KUKA KRL program: MyProgram_246().src

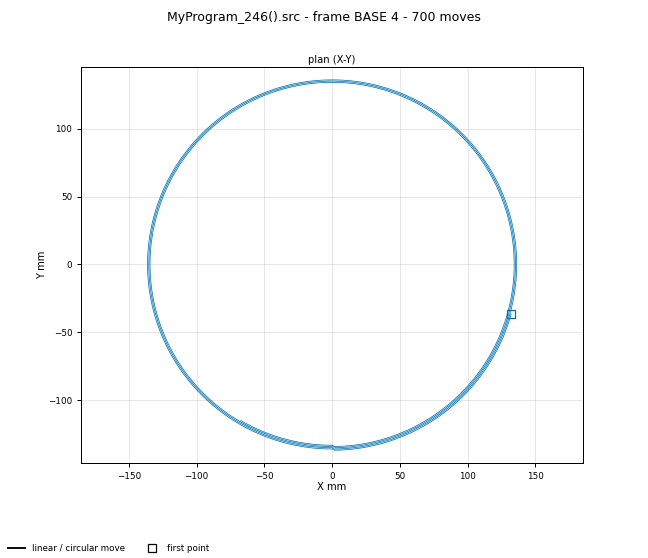
[picture p0: tool path of MyProgram_246().src in frame BASE 4, 700 of 700 moves have a stored position in this frame; points joined in program order, loops and branches not executed]
&ACCESS RVP
&REL 1
&PARAM TEMPLATE = C:\KRC\Roboter\Template\vorgabe
&PARAM EDITMASK = *
DEF MyProgram_246()
; ---- Setting reference (Base) ----
$BASE = BASE_DATA[4]

; --------------------------
; ---- Setting tool (TCP) ----
$TOOL = TOOL_DATA[3]
; --------------------------

$VEL.CP = VEL_APROX_PRINT
Startdeposition()
$VEL.CP = VEL_PRINT
LIN {X 132.0925,Y -36.5753,Z 163,A -18.1429,B 22.0609,C -0.8427,E1 22.2299,E2 825.7735} C_DIS
LIN {X 131.1106,Y -39.9509,Z 163,A -19.472,B 22.0608,C -0.8452,E1 22.2288,E2 827.0873} C_DIS
LIN {X 130.1347,Y -43.0241,Z 163,A -20.8856,B 22.061,C -0.8377,E1 22.2276,E2 828.5116} C_DIS
LIN {X 129.0285,Y -46.2357,Z 163,A -22.4856,B 22.0615,C -0.8242,E1 22.2261,E2 830.1371} C_DIS
LIN {X 126.7894,Y -52.0684,Z 163,A -24.8697,B 22.0615,C -0.8276,E1 22.2237,E2 832.4969} C_DIS
LIN {X 124.8368,Y -56.5884,Z 163,A -27.0477,B 22.0618,C -0.8153,E1 22.2212,E2 834.6937} C_DIS
LIN {X 123.0791,Y -60.313,Z 163,A -28.6428,B 22.0618,C -0.8166,E1 22.2193,E2 836.2756} C_DIS
LIN {X 121.472,Y -63.4871,Z 163,A -29.8971,B 22.0615,C -0.824,E1 22.2177,E2 837.5026} C_DIS
LIN {X 119.8871,Y -66.435,Z 163,A -31.5668,B 22.0622,C -0.8061,E1 22.2155,E2 839.2096} C_DIS
LIN {X 117.7011,Y -70.2353,Z 163,A -33.2997,B 22.0622,C -0.8059,E1 22.213,E2 840.9328} C_DIS
LIN {X 115.1668,Y -74.3185,Z 163,A -35.4245,B 22.0626,C -0.7943,E1 22.2099,E2 843.0759} C_DIS
LIN {X 113.0013,Y -77.5709,Z 163,A -36.9832,B 22.0626,C -0.7936,E1 22.2074,E2 844.6278} C_DIS
LIN {X 110.6195,Y -80.9316,Z 163,A -38.7434,B 22.0628,C -0.7869,E1 22.2045,E2 846.3958} C_DIS
LIN {X 108.0525,Y -84.3289,Z 163,A -40.5478,B 22.063,C -0.7809,E1 22.2015,E2 848.2063} C_DIS
LIN {X 105.289,Y -87.7551,Z 163,A -42.3883,B 22.0632,C -0.7761,E1 22.1982,E2 850.0499} C_DIS
LIN {X 102.3699,Y -91.1433,Z 163,A -44.2158,B 22.0632,C -0.7734,E1 22.1948,E2 851.875} C_DIS
LIN {X 99.5765,Y -94.1865,Z 163,A -45.9214,B 22.0634,C -0.7701,E1 22.1916,E2 853.5806} C_DIS
LIN {X 96.3351,Y -97.4998,Z 163,A -47.8615,B 22.0635,C -0.7653,E1 22.1878,E2 855.524} C_DIS
LIN {X 93.0592,Y -100.6314,Z 163,A -49.7722,B 22.0637,C -0.76,E1 22.1839,E2 857.4397} C_DIS
LIN {X 89.8698,Y -103.4894,Z 163,A -51.5288,B 22.0637,C -0.7576,E1 22.1802,E2 859.1947} C_DIS
LIN {X 86.486,Y -106.3335,Z 163,A -53.3585,B 22.0639,C -0.7544,E1 22.1762,E2 861.0248} C_DIS
LIN {X 82.9341,Y -109.1267,Z 163,A -55.2607,B 22.0641,C -0.7497,E1 22.172,E2 862.9314} C_DIS
LIN {X 79.2487,Y -111.8314,Z 163,A -57.1564,B 22.0641,C -0.7466,E1 22.1677,E2 864.8278} C_DIS
LIN {X 75.5656,Y -114.3522,Z 163,A -58.996,B 22.0642,C -0.7442,E1 22.1635,E2 866.6666} C_DIS
LIN {X 71.7824,Y -116.764,Z 163,A -60.8265,B 22.0642,C -0.7429,E1 22.1592,E2 868.4939} C_DIS
LIN {X 68.0323,Y -118.9881,Z 163,A -62.6432,B 22.0644,C -0.7399,E1 22.1548,E2 870.3122} C_DIS
LIN {X 64.8491,Y -120.7524,Z 163,A -64.145,B 22.0644,C -0.7382,E1 22.1511,E2 871.8134} C_DIS
LIN {X 59.748,Y -123.356,Z 163,A -66.6031,B 22.0646,C -0.7311,E1 22.1449,E2 874.2826} C_DIS
LIN {X 56.2308,Y -124.9967,Z 163,A -67.9718,B 22.0643,C -0.7412,E1 22.1415,E2 875.6207} C_DIS
LIN {X 51.2868,Y -127.105,Z 163,A -71.1817,B 22.0659,C -0.691,E1 22.1329,E2 878.9552} C_DIS
LIN {X 45.3554,Y -129.3412,Z 163,A -73.034,B 22.0648,C -0.7263,E1 22.1283,E2 880.7095} C_DIS
LIN {X 42.0092,Y -130.4659,Z 163,A -74.4413,B 22.0648,C -0.7278,E1 22.1246,E2 882.1096} C_DIS
LIN {X 38.6726,Y -131.4933,Z 163,A -75.8536,B 22.0648,C -0.7285,E1 22.1208,E2 883.5172} C_DIS
LIN {X 35.3588,Y -132.4228,Z 163,A -77.3415,B 22.0648,C -0.7246,E1 22.1168,E2 885.0128} C_DIS
LIN {X 31.7726,Y -133.3292,Z 163,A -78.9793,B 22.065,C -0.7186,E1 22.1123,E2 886.6637} C_DIS
LIN {X 27.2389,Y -134.3284,Z 163,A -81.3195,B 22.0657,C -0.6977,E1 22.1058,E2 889.0561} C_DIS
LIN {X 22.8624,Y -135.1425,Z 163,A -82.6671,B 22.065,C -0.721,E1 22.1023,E2 890.3401} C_DIS
LIN {X 19.2743,Y -135.7004,Z 163,A -84.1486,B 22.065,C -0.7217,E1 22.0982,E2 891.8181} C_DIS
LIN {X 14.7543,Y -136.266,Z 163,A -85.8072,B 22.0646,C -0.7324,E1 22.0937,E2 893.4468} C_DIS
LIN {X 8.5698,Y -136.7944,Z 163,A -88.7021,B 22.0651,C -0.7167,E1 22.0855,E2 896.3818} C_DIS
LIN {X 1.7574,Y -137.0523,Z 163,A -91.484,B 22.0651,C -0.719,E1 22.0778,E2 899.1566} C_DIS
LIN {X 1.7574,Y -137.0523,Z 163,A -91.484,B 22.0651,C -0.719,E1 22.0778,E2 899.1566} C_DIS
Enddeposition()
LIN {X 0.9573,Y -136.1368,Z 163,A -91.0711,B 20.8323,C -0.5633,E1 20.8415,E2 899.0478} C_DIS
Startdeposition()
$VEL.CP = VEL_PRINT
LIN {X 5.9809,Y -136.0119,Z 163,A -88.7973,B 20.8321,C -0.571,E1 20.8479,E2 896.7528} C_DIS
LIN {X 12.7142,Y -135.5469,Z 163,A -85.8042,B 20.8319,C -0.5792,E1 20.8563,E2 893.7385} C_DIS
LIN {X 16.2786,Y -135.1649,Z 163,A -84.4391,B 20.8321,C -0.5735,E1 20.86,E2 892.3908} C_DIS
LIN {X 19.3754,Y -134.7557,Z 163,A -83.0441,B 20.8319,C -0.578,E1 20.8639,E2 890.9845} C_DIS
LIN {X 23.679,Y -134.0667,Z 163,A -81.084,B 20.8318,C -0.5852,E1 20.8693,E2 889.007} C_DIS
LIN {X 28.5269,Y -133.1192,Z 163,A -79.1368,B 20.8318,C -0.5808,E1 20.8746,E2 887.075} C_DIS
LIN {X 31.9197,Y -132.3465,Z 163,A -77.6987,B 20.8318,C -0.581,E1 20.8785,E2 885.6389} C_DIS
LIN {X 35.3669,Y -131.4676,Z 163,A -76.2581,B 20.8319,C -0.5798,E1 20.8824,E2 884.2042} C_DIS
LIN {X 38.3717,Y -130.6219,Z 163,A -74.9511,B 20.8319,C -0.5809,E1 20.8859,E2 882.8968} C_DIS
LIN {X 41.669,Y -129.6079,Z 163,A -73.4798,B 20.8319,C -0.5835,E1 20.8899,E2 881.4216} C_DIS
LIN {X 44.6107,Y -128.6247,Z 163,A -71.8069,B 20.8313,C -0.6022,E1 20.8944,E2 879.7003} C_DIS
LIN {X 48.0166,Y -127.3927,Z 163,A -70.62,B 20.8317,C -0.5884,E1 20.8974,E2 878.5551} C_DIS
LIN {X 51.6805,Y -125.9533,Z 163,A -68.7633,B 20.8314,C -0.6,E1 20.9023,E2 876.6711} C_DIS
LIN {X 56.0611,Y -124.0638,Z 163,A -67.0228,B 20.8316,C -0.5905,E1 20.9066,E2 874.9626} C_DIS
LIN {X 59.4493,Y -122.4779,Z 163,A -65.1913,B 20.8312,C -0.605,E1 20.9113,E2 873.0964} C_DIS
LIN {X 66.6727,Y -118.7,Z 163,A -62.3065,B 20.8318,C -0.5851,E1 20.9183,E2 870.2774} C_DIS
LIN {X 70.855,Y -116.2526,Z 163,A -59.915,B 20.8312,C -0.6052,E1 20.9242,E2 867.8384} C_DIS
LIN {X 74.3486,Y -114.0495,Z 163,A -58.1316,B 20.8311,C -0.6106,E1 20.9284,E2 866.0469} C_DIS
LIN {X 78.1376,Y -111.4882,Z 163,A -56.1985,B 20.8309,C -0.6148,E1 20.9328,E2 864.1102} C_DIS
LIN {X 81.7741,Y -108.8486,Z 163,A -54.3187,B 20.8309,C -0.6181,E1 20.937,E2 862.2294} C_DIS
LIN {X 85.3978,Y -106.0291,Z 163,A -52.427,B 20.8308,C -0.6203,E1 20.9412,E2 860.3401} C_DIS
LIN {X 88.777,Y -103.2162,Z 163,A -50.5846,B 20.8307,C -0.624,E1 20.9451,E2 858.4961} C_DIS
LIN {X 92.0524,Y -100.306,Z 163,A -48.754,B 20.8306,C -0.6276,E1 20.9489,E2 856.6645} C_DIS
LIN {X 95.2418,Y -97.2828,Z 163,A -46.9125,B 20.8305,C -0.6316,E1 20.9526,E2 854.8213} C_DIS
LIN {X 98.3507,Y -94.1387,Z 163,A -45.0732,B 20.8304,C -0.6351,E1 20.9562,E2 852.9819} C_DIS
LIN {X 101.3955,Y -90.8509,Z 163,A -43.1907,B 20.8302,C -0.6396,E1 20.9597,E2 851.097} C_DIS
LIN {X 104.3997,Y -87.3822,Z 163,A -41.3152,B 20.8302,C -0.6418,E1 20.9631,E2 849.2256} C_DIS
LIN {X 107.1983,Y -83.9256,Z 163,A -39.4537,B 20.83,C -0.6462,E1 20.9664,E2 847.3625} C_DIS
LIN {X 109.7297,Y -80.5874,Z 163,A -37.6614,B 20.8299,C -0.6523,E1 20.9694,E2 845.5637} C_DIS
LIN {X 113.5217,Y -75.1515,Z 163,A -34.9433,B 20.8297,C -0.6565,E1 20.9737,E2 842.8502} C_DIS
LIN {X 117.1344,Y -69.3873,Z 163,A -32.2387,B 20.8297,C -0.6569,E1 20.9776,E2 840.1614} C_DIS
LIN {X 119.8054,Y -64.6659,Z 163,A -29.8094,B 20.8293,C -0.6705,E1 20.9809,E2 837.7095} C_DIS
LIN {X 121.5803,Y -61.2612,Z 163,A -28.2663,B 20.8293,C -0.6717,E1 20.9829,E2 836.1731} C_DIS
LIN {X 123.175,Y -57.9906,Z 163,A -26.752,B 20.8292,C -0.6754,E1 20.9847,E2 834.6584} C_DIS
LIN {X 124.9426,Y -54.0718,Z 163,A -24.9018,B 20.8289,C -0.6828,E1 20.9868,E2 832.7998} C_DIS
LIN {X 128.2312,Y -45.732,Z 163,A -21.212,B 20.8287,C -0.6902,E1 20.9905,E2 829.1146} C_DIS
LIN {X 129.623,Y -41.6217,Z 163,A -19.638,B 20.8289,C -0.6837,E1 20.9919,E2 827.5697} C_DIS
LIN {X 130.5484,Y -38.6225,Z 163,A -18.0389,B 20.8283,C -0.7011,E1 20.9932,E2 825.933} C_DIS
LIN {X 131.5669,Y -34.9944,Z 163,A -16.529,B 20.8283,C -0.7024,E1 20.9943,E2 824.43} C_DIS
LIN {X 132.5583,Y -31.0367,Z 163,A -14.8544,B 20.8282,C -0.7057,E1 20.9954,E2 822.758} C_DIS
LIN {X 133.4538,Y -26.9184,Z 163,A -13.0033,B 20.8279,C -0.7151,E1 20.9965,E2 820.894} C_DIS
LIN {X 134.2072,Y -22.8721,Z 163,A -11.2678,B 20.8277,C -0.7207,E1 20.9973,E2 819.1553} C_DIS
LIN {X 134.8677,Y -18.5875,Z 163,A -9.142,B 20.827,C -0.7411,E1 20.9982,E2 816.9878} C_DIS
LIN {X 135.323,Y -14.9104,Z 163,A -8.1608,B 20.8278,C -0.7181,E1 20.9985,E2 816.0779} C_DIS
LIN {X 135.6299,Y -11.7967,Z 163,A -6.6477,B 20.8273,C -0.7318,E1 20.9989,E2 814.5377} C_DIS
LIN {X 135.8901,Y -8.2723,Z 163,A -5.1603,B 20.8272,C -0.7366,E1 20.9992,E2 813.0477} C_DIS
LIN {X 136.1148,Y -2.7468,Z 163,A -2.7081,B 20.8267,C -0.75,E1 20.9994,E2 810.5759} C_DIS
LIN {X 136.1245,Y 2.1662,Z 163,A -0.8222,B 20.8267,C -0.7478,E1 20.9994,E2 808.7098} C_DIS
LIN {X 136.0139,Y 5.9299,Z 163,A 0.9134,B 20.8264,C -0.7601,E1 20.9992,E2 806.9525} C_DIS
LIN {X 135.735,Y 10.5321,Z 163,A 2.7811,B 20.8263,C -0.7627,E1 20.9988,E2 805.091} C_DIS
LIN {X 135.3786,Y 14.3939,Z 163,A 4.3054,B 20.8263,C -0.7627,E1 20.9984,E2 803.5778} C_DIS
LIN {X 134.9328,Y 18.1054,Z 163,A 6.012,B 20.8259,C -0.774,E1 20.9978,E2 801.8519} C_DIS
LIN {X 134.2951,Y 22.3454,Z 163,A 7.6827,B 20.8259,C -0.7732,E1 20.997,E2 800.1955} C_DIS
LIN {X 133.6398,Y 25.982,Z 163,A 9.2348,B 20.8257,C -0.7779,E1 20.9962,E2 798.6414} C_DIS
LIN {X 132.7822,Y 30.0569,Z 163,A 10.9588,B 20.8256,C -0.7819,E1 20.9952,E2 796.9185} C_DIS
LIN {X 131.9441,Y 33.5441,Z 163,A 12.4263,B 20.8255,C -0.7845,E1 20.9942,E2 795.4541} C_DIS
LIN {X 131.0161,Y 37.0048,Z 163,A 13.9109,B 20.8254,C -0.7879,E1 20.9931,E2 793.9704} C_DIS
LIN {X 129.2131,Y 42.8767,Z 163,A 16.9254,B 20.8243,C -0.8163,E1 20.9905,E2 790.8976} C_DIS
LIN {X 127.8235,Y 46.8625,Z 163,A 18.2224,B 20.825,C -0.7984,E1 20.9894,E2 789.6593} C_DIS
LIN {X 126.1483,Y 51.1969,Z 163,A 20.2191,B 20.8247,C -0.8061,E1 20.9873,E2 787.6547} C_DIS
LIN {X 124.8548,Y 54.2749,Z 163,A 21.5923,B 20.8247,C -0.8086,E1 20.9858,E2 786.2838} C_DIS
LIN {X 123.179,Y 57.9823,Z 163,A 23.3882,B 20.8243,C -0.8174,E1 20.9837,E2 784.4753} C_DIS
LIN {X 121.3746,Y 61.6653,Z 163,A 25.0582,B 20.8243,C -0.8195,E1 20.9816,E2 782.8101} C_DIS
LIN {X 119.498,Y 65.2317,Z 163,A 26.7749,B 20.824,C -0.8251,E1 20.9793,E2 781.0889} C_DIS
LIN {X 117.2985,Y 69.1089,Z 163,A 28.618,B 20.8239,C -0.8285,E1 20.9768,E2 779.2479} C_DIS
LIN {X 114.955,Y 72.9409,Z 163,A 30.4779,B 20.8237,C -0.832,E1 20.974,E2 777.3897} C_DIS
LIN {X 112.5835,Y 76.5505,Z 163,A 33.224,B 20.8218,C -0.881,E1 20.9695,E2 774.5233} C_DIS
LIN {X 108.4547,Y 82.2961,Z 163,A 35.4253,B 20.823,C -0.8512,E1 20.966,E2 772.4183} C_DIS
LIN {X 105.3366,Y 86.2504,Z 163,A 37.38,B 20.8231,C -0.8484,E1 20.9626,E2 770.4824} C_DIS
LIN {X 102.4793,Y 89.6268,Z 163,A 39.4353,B 20.8226,C -0.8619,E1 20.9588,E2 768.401} C_DIS
LIN {X 100.3058,Y 92.0526,Z 163,A 40.4025,B 20.8232,C -0.846,E1 20.9571,E2 767.4835} C_DIS
LIN {X 98.0621,Y 94.4398,Z 163,A 41.985,B 20.8227,C -0.8585,E1 20.954,E2 765.8743} C_DIS
LIN {X 94.9308,Y 97.5868,Z 163,A 43.8663,B 20.8225,C -0.8631,E1 20.9502,E2 763.9898} C_DIS
LIN {X 91.9581,Y 100.3927,Z 163,A 45.5187,B 20.8225,C -0.8634,E1 20.9469,E2 762.3448} C_DIS
LIN {X 88.7505,Y 103.239,Z 163,A 48.4672,B 20.8202,C -0.9208,E1 20.9403,E2 759.2496} C_DIS
LIN {X 82.3061,Y 108.4471,Z 163,A 50.5399,B 20.8226,C -0.8608,E1 20.9361,E2 757.3544} C_DIS
LIN {X 79.4229,Y 110.5759,Z 163,A 52.2003,B 20.8222,C -0.8705,E1 20.9323,E2 755.6742} C_DIS
LIN {X 76.1216,Y 112.8738,Z 163,A 53.9563,B 20.822,C -0.8762,E1 20.9283,E2 753.9094} C_DIS
LIN {X 72.4598,Y 115.2587,Z 163,A 55.8307,B 20.8218,C -0.8807,E1 20.9238,E2 752.0297} C_DIS
LIN {X 68.6015,Y 117.5965,Z 163,A 57.7104,B 20.8218,C -0.8827,E1 20.9193,E2 750.1516} C_DIS
LIN {X 64.807,Y 119.7296,Z 163,A 59.5703,B 20.8216,C -0.8865,E1 20.9148,E2 748.2876} C_DIS
LIN {X 61.5076,Y 121.4549,Z 163,A 61.0638,B 20.8216,C -0.8853,E1 20.9111,E2 746.8028} C_DIS
LIN {X 57.8827,Y 123.2261,Z 163,A 62.8484,B 20.8214,C -0.8913,E1 20.9066,E2 745.007} C_DIS
LIN {X 53.4721,Y 125.2019,Z 163,A 64.7371,B 20.8216,C -0.887,E1 20.9018,E2 743.136} C_DIS
LIN {X 47.2983,Y 127.6618,Z 163,A 67.0639,B 20.8223,C -0.8685,E1 20.8959,E2 740.8675} C_DIS
LIN {X 44.4361,Y 128.6852,Z 163,A 68.7845,B 20.8215,C -0.8896,E1 20.8912,E2 739.092} C_DIS
LIN {X 41.1735,Y 129.7661,Z 163,A 70.2438,B 20.8214,C -0.8914,E1 20.8873,E2 737.631} C_DIS
LIN {X 38.008,Y 130.7284,Z 163,A 71.6147,B 20.8214,C -0.8914,E1 20.8837,E2 736.2629} C_DIS
LIN {X 34.8398,Y 131.6081,Z 163,A 73.039,B 20.8213,C -0.8942,E1 20.8798,E2 734.8335} C_DIS
LIN {X 30.6655,Y 132.6432,Z 163,A 74.8681,B 20.8212,C -0.8961,E1 20.8748,E2 733.0023} C_DIS
LIN {X 26.8947,Y 133.4587,Z 163,A 76.4627,B 20.8212,C -0.8956,E1 20.8705,E2 731.4115} C_DIS
LIN {X 21.3324,Y 134.4607,Z 163,A 78.6958,B 20.8214,C -0.89,E1 20.8644,E2 729.1971} C_DIS
LIN {X 17.5624,Y 135.004,Z 163,A 80.4262,B 20.8212,C -0.8962,E1 20.8596,E2 727.4513} C_DIS
LIN {X 13.5394,Y 135.4677,Z 163,A 82.3449,B 20.8208,C -0.906,E1 20.8542,E2 725.5065} C_DIS
LIN {X 7.7658,Y 135.9213,Z 163,A 84.5265,B 20.8212,C -0.8948,E1 20.8482,E2 723.3577} C_DIS
LIN {X 4.097,Y 136.0804,Z 163,A 86.1427,B 20.8212,C -0.8979,E1 20.8437,E2 721.7334} C_DIS
LIN {X 0.3597,Y 136.1418,Z 163,A 87.9402,B 20.8207,C -0.9076,E1 20.8386,E2 719.9086} C_DIS
LIN {X -5.8293,Y 136.0178,Z 163,A 90.4101,B 20.821,C -0.901,E1 20.8317,E2 717.457} C_DIS
LIN {X -9.9412,Y 135.7781,Z 163,A 91.9998,B 20.8213,C -0.8941,E1 20.8273,E2 715.8861} C_DIS
LIN {X -13.4121,Y 135.4799,Z 163,A 93.6793,B 20.8209,C -0.9028,E1 20.8226,E2 714.1811} C_DIS
LIN {X -17.2844,Y 135.0404,Z 163,A 95.1442,B 20.8213,C -0.8942,E1 20.8186,E2 712.7391} C_DIS
LIN {X -20.8954,Y 134.5284,Z 163,A 96.7643,B 20.8212,C -0.897,E1 20.8141,E2 711.1095} C_DIS
LIN {X -24.8379,Y 133.8585,Z 163,A 98.5198,B 20.8211,C -0.8989,E1 20.8093,E2 709.3464} C_DIS
LIN {X -29.0692,Y 133.0022,Z 163,A 100.138,B 20.8215,C -0.8888,E1 20.8049,E2 707.7542} C_DIS
LIN {X -32.1683,Y 132.2866,Z 163,A 101.5117,B 20.8215,C -0.8892,E1 20.8012,E2 706.3773} C_DIS
LIN {X -35.917,Y 131.3203,Z 163,A 103.8019,B 20.8204,C -0.9163,E1 20.7948,E2 704.0064} C_DIS
LIN {X -40.8106,Y 129.8821,Z 163,A 105.2335,B 20.8217,C -0.8829,E1 20.7912,E2 702.6659} C_DIS
LIN {X -44.8032,Y 128.5579,Z 163,A 107.097,B 20.8217,C -0.8849,E1 20.7862,E2 700.7924} C_DIS
LIN {X -48.3813,Y 127.2561,Z 163,A 109.0164,B 20.8212,C -0.8965,E1 20.7811,E2 698.8355} C_DIS
LIN {X -51.5758,Y 125.9954,Z 163,A 110.1213,B 20.8219,C -0.8799,E1 20.7784,E2 697.7743} C_DIS
LIN {X -54.4325,Y 124.7866,Z 163,A 111.4691,B 20.8219,C -0.8799,E1 20.7749,E2 696.4227} C_DIS
LIN {X -57.5838,Y 123.3643,Z 163,A 113.0577,B 20.8217,C -0.8835,E1 20.7708,E2 694.8192} C_DIS
LIN {X -61.7482,Y 121.3324,Z 163,A 114.8859,B 20.822,C -0.8753,E1 20.7663,E2 693.0083} C_DIS
LIN {X -66.637,Y 118.72,Z 163,A 117.2559,B 20.8221,C -0.873,E1 20.7605,E2 690.6366} C_DIS
LIN {X -70.2398,Y 116.6249,Z 163,A 119.0789,B 20.8221,C -0.8728,E1 20.7561,E2 688.8073} C_DIS
LIN {X -74.0171,Y 114.2647,Z 163,A 121.0574,B 20.8221,C -0.8738,E1 20.7514,E2 686.8183} C_DIS
LIN {X -77.6596,Y 111.8207,Z 163,A 122.9462,B 20.8221,C -0.872,E1 20.7471,E2 684.9266} C_DIS
LIN {X -81.7195,Y 108.8897,Z 163,A 124.9509,B 20.8225,C -0.8634,E1 20.7426,E2 682.9375} C_DIS
LIN {X -85.1756,Y 106.2083,Z 163,A 126.7323,B 20.8228,C -0.8571,E1 20.7387,E2 681.166} C_DIS
LIN {X -88.4711,Y 103.4792,Z 163,A 128.6154,B 20.8228,C -0.8566,E1 20.7347,E2 679.2753} C_DIS
LIN {X -91.8613,Y 100.4817,Z 163,A 130.5003,B 20.823,C -0.8515,E1 20.7308,E2 677.3955} C_DIS
LIN {X -95.0379,Y 97.4828,Z 163,A 132.3997,B 20.823,C -0.8498,E1 20.7269,E2 675.4914} C_DIS
LIN {X -98.2023,Y 94.2939,Z 163,A 134.2528,B 20.8233,C -0.8437,E1 20.7233,E2 673.6457} C_DIS
LIN {X -101.1802,Y 91.0913,Z 163,A 136.1455,B 20.8233,C -0.8414,E1 20.7198,E2 671.7494} C_DIS
LIN {X -105.6974,Y 85.808,Z 163,A 139.025,B 20.8237,C -0.8321,E1 20.7146,E2 668.8801} C_DIS
LIN {X -110.6727,Y 79.2874,Z 163,A 142.9014,B 20.8234,C -0.8406,E1 20.7081,E2 664.9567} C_DIS
LIN {X -113.073,Y 75.8256,Z 163,A 144.0969,B 20.8245,C -0.8118,E1 20.7063,E2 663.8354} C_DIS
LIN {X -114.6408,Y 73.4331,Z 163,A 145.505,B 20.8243,C -0.8169,E1 20.7041,E2 662.4041} C_DIS
LIN {X -117.0187,Y 69.5814,Z 163,A 147.4308,B 20.8245,C -0.8124,E1 20.7014,E2 660.4789} C_DIS
LIN {X -120.983,Y 62.4345,Z 163,A 151.1407,B 20.8245,C -0.8137,E1 20.6964,E2 656.7413} C_DIS
LIN {X -122.5226,Y 59.3561,Z 163,A 152.23,B 20.8251,C -0.7946,E1 20.6951,E2 655.6989} C_DIS
LIN {X -123.6631,Y 56.9376,Z 163,A 153.4169,B 20.8251,C -0.7938,E1 20.6937,E2 654.5062} C_DIS
LIN {X -125.2267,Y 53.4145,Z 163,A 155.2445,B 20.8251,C -0.7975,E1 20.6917,E2 652.6559} C_DIS
LIN {X -126.8586,Y 49.4097,Z 163,A 156.9217,B 20.8254,C -0.7861,E1 20.69,E2 650.9994} C_DIS
LIN {X -128.251,Y 45.6769,Z 163,A 158.6773,B 20.8255,C -0.7842,E1 20.6883,E2 649.2369} C_DIS
LIN {X -129.6144,Y 41.6485,Z 163,A 160.3687,B 20.8258,C -0.7747,E1 20.6868,E2 647.5607} C_DIS
LIN {X -130.7959,Y 37.7774,Z 163,A 162.076,B 20.826,C -0.7696,E1 20.6854,E2 645.8557} C_DIS
LIN {X -131.5688,Y 34.9873,Z 163,A 163.3057,B 20.8261,C -0.7663,E1 20.6846,E2 644.6267} C_DIS
LIN {X -132.4179,Y 31.6236,Z 163,A 164.8344,B 20.8262,C -0.7645,E1 20.6835,E2 643.092} C_DIS
LIN {X -133.3651,Y 27.3547,Z 163,A 166.6594,B 20.8264,C -0.7581,E1 20.6825,E2 641.2719} C_DIS
LIN {X -134.0485,Y 23.781,Z 163,A 168.159,B 20.8266,C -0.752,E1 20.6817,E2 639.7788} C_DIS
LIN {X -134.5945,Y 20.4685,Z 163,A 169.7405,B 20.8266,C -0.7544,E1 20.681,E2 638.1788} C_DIS
LIN {X -135.1778,Y 16.1699,Z 163,A 171.4502,B 20.8269,C -0.7439,E1 20.6804,E2 636.4865} C_DIS
LIN {X -135.5459,Y 12.724,Z 163,A 172.9275,B 20.8271,C -0.74,E1 20.68,E2 635.0093} C_DIS
LIN {X -135.8612,Y 8.7417,Z 163,A 174.6666,B 20.8271,C -0.737,E1 20.6797,E2 633.2658} C_DIS
LIN {X -136.0416,Y 5.2189,Z 163,A 176.1221,B 20.8274,C -0.7311,E1 20.6795,E2 631.8163} C_DIS
LIN {X -136.136,Y 1.4189,Z 163,A 177.7923,B 20.8274,C -0.7289,E1 20.6795,E2 630.14} C_DIS
LIN {X -136.1117,Y -2.9358,Z 163,A 179.6957,B 20.8275,C -0.726,E1 20.6795,E2 628.2307} C_DIS
LIN {X -135.9626,Y -6.9812,Z 163,A -178.7261,B 20.8279,C -0.7155,E1 20.6797,E2 626.6708} C_DIS
LIN {X -135.7132,Y -10.8108,Z 163,A -176.9918,B 20.8279,C -0.7153,E1 20.68,E2 624.9243} C_DIS
LIN {X -135.3431,Y -14.7234,Z 163,A -175.4203,B 20.8282,C -0.7067,E1 20.6805,E2 623.3656} C_DIS
LIN {X -134.8365,Y -18.8103,Z 163,A -173.6236,B 20.8282,C -0.7039,E1 20.6811,E2 621.5636} C_DIS
LIN {X -134.2924,Y -22.3615,Z 163,A -172.1656,B 20.8285,C -0.6969,E1 20.6818,E2 620.1146} C_DIS
LIN {X -133.6825,Y -25.7585,Z 163,A -170.7234,B 20.8286,C -0.692,E1 20.6825,E2 618.6759} C_DIS
LIN {X -133.0247,Y -28.9648,Z 163,A -169.2852,B 20.8286,C -0.6903,E1 20.6833,E2 617.2321} C_DIS
LIN {X -132.2792,Y -32.1988,Z 163,A -167.8427,B 20.8288,C -0.6879,E1 20.6843,E2 615.786} C_DIS
LIN {X -130.7052,Y -38.0869,Z 163,A -165.5601,B 20.8294,C -0.6685,E1 20.6859,E2 613.5422} C_DIS
LIN {X -129.6447,Y -41.5536,Z 163,A -163.7493,B 20.8291,C -0.6757,E1 20.6874,E2 611.6981} C_DIS
LIN {X -128.5232,Y -44.9034,Z 163,A -162.3055,B 20.8293,C -0.6696,E1 20.6887,E2 610.2616} C_DIS
LIN {X -127.4779,Y -47.7891,Z 163,A -160.9544,B 20.8293,C -0.6683,E1 20.69,E2 608.9048} C_DIS
LIN {X -126.1781,Y -51.1229,Z 163,A -159.4282,B 20.8295,C -0.6648,E1 20.6916,E2 607.3782} C_DIS
LIN {X -124.5868,Y -54.8918,Z 163,A -156.808,B 20.8285,C -0.6976,E1 20.6947,E2 604.6472} C_DIS
LIN {X -121.8227,Y -60.7783,Z 163,A -154.9709,B 20.8299,C -0.6521,E1 20.6968,E2 602.9269} C_DIS
LIN {X -120.2522,Y -63.8291,Z 163,A -153.3683,B 20.8298,C -0.6548,E1 20.6989,E2 601.3062} C_DIS
LIN {X -118.4363,Y -67.141,Z 163,A -151.7764,B 20.8299,C -0.6506,E1 20.7011,E2 599.7158} C_DIS
LIN {X -116.1072,Y -71.092,Z 163,A -149.8622,B 20.8301,C -0.6449,E1 20.7038,E2 597.8058} C_DIS
LIN {X -113.7371,Y -74.8252,Z 163,A -147.8731,B 20.8301,C -0.6455,E1 20.7069,E2 595.8027} C_DIS
LIN {X -111.2507,Y -78.4743,Z 163,A -146.1168,B 20.8303,C -0.6365,E1 20.7097,E2 594.0611} C_DIS
LIN {X -108.5291,Y -82.1975,Z 163,A -144.137,B 20.8304,C -0.6334,E1 20.713,E2 592.0784} C_DIS
LIN {X -105.6584,Y -85.8567,Z 163,A -142.225,B 20.8306,C -0.6269,E1 20.7163,E2 590.1739} C_DIS
LIN {X -102.7115,Y -89.3606,Z 163,A -140.4717,B 20.8309,C -0.6151,E1 20.7194,E2 588.4442} C_DIS
LIN {X -100.6359,Y -91.692,Z 163,A -138.9687,B 20.8308,C -0.6202,E1 20.7223,E2 586.9185} C_DIS
LIN {X -97.6641,Y -94.8509,Z 163,A -137.1109,B 20.8308,C -0.6176,E1 20.7259,E2 585.0581} C_DIS
LIN {X -94.4263,Y -98.0752,Z 163,A -135.1682,B 20.831,C -0.6144,E1 20.7297,E2 583.1144} C_DIS
LIN {X -91.1334,Y -101.1424,Z 163,A -132.6379,B 20.8303,C -0.6381,E1 20.7352,E2 580.5049} C_DIS
LIN {X -86.9261,Y -104.7798,Z 163,A -130.9172,B 20.8312,C -0.6068,E1 20.7387,E2 578.8644} C_DIS
LIN {X -83.3708,Y -107.6301,Z 163,A -128.889,B 20.8312,C -0.6081,E1 20.7431,E2 576.8234} C_DIS
LIN {X -79.4778,Y -110.5366,Z 163,A -126.9727,B 20.8314,C -0.599,E1 20.7474,E2 574.9244} C_DIS
LIN {X -75.9559,Y -112.986,Z 163,A -125.0987,B 20.8314,C -0.599,E1 20.7517,E2 573.0428} C_DIS
LIN {X -72.2627,Y -115.3828,Z 163,A -123.239,B 20.8314,C -0.5965,E1 20.7561,E2 571.183} C_DIS
LIN {X -68.5357,Y -117.6348,Z 163,A -121.4131,B 20.8315,C -0.5935,E1 20.7605,E2 569.3587} C_DIS
LIN {X -64.7496,Y -119.7604,Z 163,A -119.5834,B 20.8315,C -0.5911,E1 20.765,E2 567.5293} C_DIS
LIN {X -61.4846,Y -121.4666,Z 163,A -118.1403,B 20.8318,C -0.5845,E1 20.7685,E2 566.1001} C_DIS
LIN {X -58.733,Y -122.8203,Z 163,A -116.766,B 20.8318,C -0.5866,E1 20.772,E2 564.7155} C_DIS
LIN {X -54.9297,Y -124.5699,Z 163,A -114.3782,B 20.831,C -0.6122,E1 20.7783,E2 562.2485} C_DIS
LIN {X -49.9485,Y -126.6492,Z 163,A -112.8635,B 20.832,C -0.5765,E1 20.782,E2 560.8305} C_DIS
LIN {X -45.0737,Y -128.4642,Z 163,A -110.5012,B 20.8318,C -0.5821,E1 20.7882,E2 558.4465} C_DIS
LIN {X -41.3262,Y -129.7173,Z 163,A -108.9279,B 20.832,C -0.5768,E1 20.7924,E2 556.8845} C_DIS
LIN {X -38.1106,Y -130.6983,Z 163,A -107.5176,B 20.832,C -0.5756,E1 20.7962,E2 555.4748} C_DIS
LIN {X -34.8818,Y -131.5969,Z 163,A -106.1032,B 20.832,C -0.5749,E1 20.8,E2 554.0599} C_DIS
LIN {X -31.3815,Y -132.4762,Z 163,A -104.6066,B 20.832,C -0.573,E1 20.804,E2 552.5659} C_DIS
LIN {X -28.0033,Y -133.2323,Z 163,A -102.607,B 20.8314,C -0.5966,E1 20.8097,E2 550.4969} C_DIS
LIN {X -23.7225,Y -134.0589,Z 163,A -101.4698,B 20.8323,C -0.5647,E1 20.8126,E2 549.4482} C_DIS
LIN {X -20.8214,Y -134.5398,Z 163,A -100.0094,B 20.832,C -0.5742,E1 20.8167,E2 547.9593} C_DIS
LIN {X -16.5914,Y -135.1275,Z 163,A -97.9491,B 20.8317,C -0.5857,E1 20.8225,E2 545.8651} C_DIS
LIN {X -13.3298,Y -135.4878,Z 163,A -96.2394,B 20.8313,C -0.6004,E1 20.8273,E2 544.1126} C_DIS
LIN {X -8.2889,Y -135.8891,Z 163,A -94.733,B 20.8321,C -0.5722,E1 20.8313,E2 542.6851} C_DIS
LIN {X -4.6976,Y -136.0619,Z 163,A -92.5718,B 20.8313,C -0.6018,E1 20.8376,E2 540.4403} C_DIS
LIN {X 0.4637,Y -136.1412,Z 163,A -91.0917,B 20.8321,C -0.5707,E1 20.8415,E2 539.0478} C_DIS
LIN {X 0.4637,Y -136.1412,Z 163,A -91.0917,B 20.8321,C -0.5707,E1 20.8415,E2 539.0478} C_DIS
Enddeposition()
LIN {X 0.9493,Y -135.2146,Z 163,A -90.7114,B 19.607,C -0.4067,E1 19.6129,E2 539.0313} C_DIS
Startdeposition()
$VEL.CP = VEL_PRINT
LIN {X -2.1021,Y -135.2045,Z 163,A -92.3957,B 19.6073,C -0.39,E1 19.6081,E2 540.7652} C_DIS
LIN {X -5.3088,Y -135.1165,Z 163,A -93.7552,B 19.6073,C -0.3899,E1 19.6043,E2 542.1254} C_DIS
LIN {X -9.0786,Y -134.9177,Z 163,A -95.339,B 19.6073,C -0.3905,E1 19.5999,E2 543.708} C_DIS
LIN {X -13.0731,Y -134.5873,Z 163,A -97.0415,B 19.6073,C -0.3905,E1 19.5951,E2 545.4115} C_DIS
LIN {X -16.1777,Y -134.2494,Z 163,A -98.3767,B 19.6073,C -0.3902,E1 19.5914,E2 546.7486} C_DIS
LIN {X -19.44,Y -133.8162,Z 163,A -99.8068,B 19.6073,C -0.3891,E1 19.5874,E2 548.1836} C_DIS
LIN {X -23.0371,Y -133.246,Z 163,A -101.3121,B 19.6073,C -0.3911,E1 19.5833,E2 549.6846} C_DIS
LIN {X -27.1167,Y -132.4737,Z 163,A -103.0903,B 19.6073,C -0.3911,E1 19.5784,E2 551.4654} C_DIS
LIN {X -30.8991,Y -131.6452,Z 163,A -104.7215,B 19.6073,C -0.3923,E1 19.574,E2 553.0958} C_DIS
LIN {X -34.053,Y -130.8649,Z 163,A -106.1025,B 19.6073,C -0.3929,E1 19.5702,E2 554.4774} C_DIS
LIN {X -36.7609,Y -130.128,Z 163,A -107.3146,B 19.6073,C -0.3929,E1 19.567,E2 555.6924} C_DIS
LIN {X -39.9661,Y -129.1798,Z 163,A -108.7479,B 19.6073,C -0.3932,E1 19.5631,E2 557.1278} C_DIS
LIN {X -43.5078,Y -128.0324,Z 163,A -110.2993,B 19.6072,C -0.3955,E1 19.559,E2 558.676} C_DIS
LIN {X -46.647,Y -126.9223,Z 163,A -111.7153,B 19.6072,C -0.3965,E1 19.5553,E2 560.0927} C_DIS
LIN {X -49.2925,Y -125.9161,Z 163,A -112.9656,B 19.6072,C -0.3956,E1 19.552,E2 561.349} C_DIS
LIN {X -52.888,Y -124.4511,Z 163,A -114.5705,B 19.6072,C -0.3989,E1 19.5479,E2 562.9489} C_DIS
LIN {X -55.9833,Y -123.0898,Z 163,A -116.009,B 19.6072,C -0.4003,E1 19.5442,E2 564.3878} C_DIS
LIN {X -58.6845,Y -121.8229,Z 163,A -117.3093,B 19.6072,C -0.4003,E1 19.5409,E2 565.6922} C_DIS
LIN {X -62.1071,Y -120.1163,Z 163,A -118.9059,B 19.607,C -0.4033,E1 19.537,E2 567.2856} C_DIS
LIN {X -64.8264,Y -118.67,Z 163,A -120.2658,B 19.607,C -0.4029,E1 19.5336,E2 568.6518} C_DIS
LIN {X -68.5638,Y -116.5506,Z 163,A -122.0948,B 19.607,C -0.4051,E1 19.5292,E2 570.4812} C_DIS
LIN {X -72.2468,Y -114.3041,Z 163,A -123.9267,B 19.607,C -0.4077,E1 19.5248,E2 572.3129} C_DIS
LIN {X -75.6611,Y -112.0735,Z 163,A -125.7191,B 19.607,C -0.4079,E1 19.5207,E2 574.1125} C_DIS
LIN {X -79.4241,Y -109.4388,Z 163,A -127.6243,B 19.6069,C -0.4128,E1 19.5163,E2 576.0117} C_DIS
LIN {X -82.906,Y -106.8252,Z 163,A -129.4785,B 19.6068,C -0.4156,E1 19.5122,E2 577.8661} C_DIS
LIN {X -86.3088,Y -104.0953,Z 163,A -131.3367,B 19.6068,C -0.4187,E1 19.5082,E2 579.7244} C_DIS
LIN {X -89.6267,Y -101.2526,Z 163,A -133.1979,B 19.6067,C -0.4218,E1 19.5043,E2 581.5856} C_DIS
LIN {X -92.7965,Y -98.3556,Z 163,A -135.0426,B 19.6067,C -0.4245,E1 19.5005,E2 583.4322} C_DIS
LIN {X -95.8341,Y -95.3985,Z 163,A -136.8771,B 19.6066,C -0.4267,E1 19.4968,E2 585.27} C_DIS
LIN {X -98.9001,Y -92.2161,Z 163,A -138.7508,B 19.6065,C -0.4307,E1 19.4932,E2 587.1425} C_DIS
LIN {X -101.83,Y -88.9702,Z 163,A -140.6142,B 19.6065,C -0.4344,E1 19.4898,E2 589.0057} C_DIS
LIN {X -104.6504,Y -85.6349,Z 163,A -142.4758,B 19.6063,C -0.4383,E1 19.4865,E2 590.8669} C_DIS
LIN {X -107.461,Y -82.0803,Z 163,A -144.3614,B 19.6062,C -0.4442,E1 19.4832,E2 592.7466} C_DIS
LIN {X -109.9472,Y -78.7187,Z 163,A -146.1894,B 19.6062,C -0.4463,E1 19.4802,E2 594.5798} C_DIS
LIN {X -112.5111,Y -75.0086,Z 163,A -148.0785,B 19.606,C -0.4519,E1 19.4773,E2 596.4644} C_DIS
LIN {X -114.8253,Y -71.4156,Z 163,A -149.9023,B 19.606,C -0.4561,E1 19.4745,E2 598.2879} C_DIS
LIN {X -116.9847,Y -67.8205,Z 163,A -151.7216,B 19.6059,C -0.4591,E1 19.4719,E2 600.1105} C_DIS
LIN {X -119.0456,Y -64.1342,Z 163,A -153.5371,B 19.6058,C -0.4629,E1 19.4695,E2 601.9271} C_DIS
LIN {X -120.8909,Y -60.5855,Z 163,A -155.1456,B 19.6056,C -0.4708,E1 19.4675,E2 603.5232} C_DIS
LIN {X -122.3777,Y -57.5232,Z 163,A -156.5972,B 19.6056,C -0.4744,E1 19.4657,E2 604.9743} C_DIS
LIN {X -123.7809,Y -54.4381,Z 163,A -158.0426,B 19.6054,C -0.478,E1 19.4641,E2 606.419} C_DIS
LIN {X -124.9644,Y -51.6588,Z 163,A -159.3539,B 19.6054,C -0.4805,E1 19.4627,E2 607.7325} C_DIS
LIN {X -126.3359,Y -48.2125,Z 163,A -160.9127,B 19.6053,C -0.4855,E1 19.4611,E2 609.2879} C_DIS
LIN {X -127.3024,Y -45.5929,Z 163,A -162.1363,B 19.6053,C -0.4874,E1 19.4599,E2 610.5148} C_DIS
LIN {X -128.5562,Y -41.9349,Z 163,A -163.7529,B 19.6051,C -0.493,E1 19.4585,E2 612.1267} C_DIS
LIN {X -129.5414,Y -38.7844,Z 163,A -165.1609,B 19.605,C -0.4967,E1 19.4573,E2 613.534} C_DIS
LIN {X -130.4442,Y -35.6304,Z 163,A -166.5598,B 19.6049,C -0.5005,E1 19.4563,E2 614.9322} C_DIS
LIN {X -131.2652,Y -32.4757,Z 163,A -167.9502,B 19.6048,C -0.5043,E1 19.4553,E2 616.3218} C_DIS
LIN {X -132.0051,Y -29.3234,Z 163,A -169.3309,B 19.6048,C -0.5082,E1 19.4545,E2 617.7017} C_DIS
LIN {X -132.6651,Y -26.1763,Z 163,A -170.7027,B 19.6046,C -0.512,E1 19.4537,E2 619.0726} C_DIS
LIN {X -133.2166,Y -23.2015,Z 163,A -171.9658,B 19.6045,C -0.5166,E1 19.4531,E2 620.3316} C_DIS
LIN {X -133.6748,Y -20.3894,Z 163,A -173.2514,B 19.6045,C -0.5174,E1 19.4525,E2 621.625} C_DIS
LIN {X -134.176,Y -16.7933,Z 163,A -174.7565,B 19.6043,C -0.5234,E1 19.452,E2 623.1238} C_DIS
LIN {X -134.5277,Y -13.6936,Z 163,A -176.0871,B 19.6043,C -0.5271,E1 19.4516,E2 624.4536} C_DIS
LIN {X -134.839,Y -10.1569,Z 163,A -177.6612,B 19.6042,C -0.5292,E1 19.4512,E2 626.0338} C_DIS
LIN {X -135.0606,Y -6.5808,Z 163,A -179.12,B 19.604,C -0.5362,E1 19.451,E2 627.4831} C_DIS
LIN {X -135.1895,Y -3.0014,Z 163,A 179.3433,B 19.6039,C -0.5402,E1 19.4508,E2 629.0199} C_DIS
LIN {X -135.2202,Y 0.6542,Z 163,A 177.7306,B 19.6039,C -0.5427,E1 19.4508,E2 630.6379} C_DIS
LIN {X -135.1644,Y 3.9045,Z 163,A 176.3231,B 19.6037,C -0.5459,E1 19.4509,E2 632.0469} C_DIS
LIN {X -135.0426,Y 6.9385,Z 163,A 175.0225,B 19.6037,C -0.5494,E1 19.4511,E2 633.3472} C_DIS
LIN {X -134.8058,Y 10.612,Z 163,A 173.5146,B 19.6034,C -0.5562,E1 19.4514,E2 634.8465} C_DIS
LIN {X -134.4281,Y 14.619,Z 163,A 171.7711,B 19.6034,C -0.5602,E1 19.4519,E2 636.5918} C_DIS
LIN {X -134.0294,Y 17.9123,Z 163,A 170.3943,B 19.6032,C -0.5657,E1 19.4524,E2 637.9629} C_DIS
LIN {X -133.5805,Y 20.9988,Z 163,A 169.0391,B 19.6032,C -0.5685,E1 19.4529,E2 639.3201} C_DIS
LIN {X -132.9653,Y 24.6056,Z 163,A 167.4707,B 19.603,C -0.5727,E1 19.4537,E2 640.8883} C_DIS
LIN {X -132.345,Y 27.749,Z 163,A 166.0993,B 19.6029,C -0.5764,E1 19.4544,E2 642.2592} C_DIS
LIN {X -131.418,Y 31.8418,Z 163,A 164.2848,B 19.6028,C -0.5805,E1 19.4556,E2 644.0752} C_DIS
LIN {X -130.4442,Y 35.6304,Z 163,A 162.6299,B 19.6026,C -0.5857,E1 19.4568,E2 645.7272} C_DIS
LIN {X -129.5414,Y 38.7844,Z 163,A 161.2267,B 19.6026,C -0.5895,E1 19.4579,E2 647.1297} C_DIS
LIN {X -128.5562,Y 41.9349,Z 163,A 159.8147,B 19.6024,C -0.5932,E1 19.4591,E2 648.5411} C_DIS
LIN {X -127.6112,Y 44.7227,Z 163,A 158.5289,B 19.6024,C -0.5955,E1 19.4602,E2 649.8294} C_DIS
LIN {X -126.3359,Y 48.2125,Z 163,A 156.9671,B 19.6022,C -0.6007,E1 19.4618,E2 651.3874} C_DIS
LIN {X -125.1003,Y 51.3334,Z 163,A 155.5317,B 19.6021,C -0.6044,E1 19.4633,E2 652.8221} C_DIS
LIN {X -123.8907,Y 54.184,Z 163,A 154.219,B 19.602,C -0.6083,E1 19.4647,E2 654.1326} C_DIS
LIN {X -122.3777,Y 57.5232,Z 163,A 152.6408,B 19.6019,C -0.6119,E1 19.4665,E2 655.7115} C_DIS
LIN {X -120.8909,Y 60.5855,Z 163,A 151.1859,B 19.6017,C -0.6155,E1 19.4683,E2 657.1656} C_DIS
LIN {X -119.3209,Y 63.6218,Z 163,A 149.7664,B 19.6016,C -0.6208,E1 19.4702,E2 658.5793} C_DIS
LIN {X -117.6684,Y 66.6286,Z 163,A 148.1461,B 19.6016,C -0.6186,E1 19.4724,E2 660.2174} C_DIS
LIN {X -115.4877,Y 70.3407,Z 163,A 146.3066,B 19.6016,C -0.623,E1 19.475,E2 662.0559} C_DIS
LIN {X -113.1809,Y 73.9953,Z 163,A 144.4915,B 19.6013,C -0.6286,E1 19.4778,E2 663.8662} C_DIS
LIN {X -110.7503,Y 77.586,Z 163,A 142.6404,B 19.6013,C -0.633,E1 19.4807,E2 665.7161} C_DIS
LIN {X -108.1985,Y 81.1068,Z 163,A 140.7523,B 19.6011,C -0.6361,E1 19.4838,E2 667.6069} C_DIS
LIN {X -105.5285,Y 84.5514,Z 163,A 138.892,B 19.601,C -0.6403,E1 19.487,E2 669.4661} C_DIS
LIN {X -102.744,Y 87.9141,Z 163,A 137.0634,B 19.6008,C -0.6457,E1 19.4903,E2 671.2893} C_DIS
LIN {X -99.8486,Y 91.1892,Z 163,A 135.1642,B 19.6008,C -0.6485,E1 19.4939,E2 673.1915} C_DIS
LIN {X -96.8466,Y 94.3713,Z 163,A 133.3301,B 19.6006,C -0.6536,E1 19.4974,E2 675.0206} C_DIS
LIN {X -93.7426,Y 97.4553,Z 163,A 131.4712,B 19.6004,C -0.6577,E1 19.5011,E2 676.8775} C_DIS
LIN {X -90.5415,Y 100.4363,Z 163,A 129.6004,B 19.6004,C -0.6611,E1 19.505,E2 678.7477} C_DIS
LIN {X -87.2484,Y 103.3099,Z 163,A 127.7382,B 19.6002,C -0.6647,E1 19.5089,E2 680.6086} C_DIS
LIN {X -83.8689,Y 106.0718,Z 163,A 125.8481,B 19.6002,C -0.667,E1 19.513,E2 682.5011} C_DIS
LIN {X -80.4085,Y 108.7184,Z 163,A 124.0244,B 19.6,C -0.6716,E1 19.5171,E2 684.3198} C_DIS
LIN {X -76.8733,Y 111.2462,Z 163,A 122.1436,B 19.6,C -0.6736,E1 19.5214,E2 686.2029} C_DIS
LIN {X -73.2692,Y 113.6522,Z 163,A 120.2999,B 19.5998,C -0.6767,E1 19.5257,E2 688.0453} C_DIS
LIN {X -69.6026,Y 115.934,Z 163,A 118.4937,B 19.5997,C -0.6808,E1 19.53,E2 689.8464} C_DIS
LIN {X -65.8798,Y 118.0892,Z 163,A 116.6339,B 19.5997,C -0.6824,E1 19.5345,E2 691.7085} C_DIS
LIN {X -62.1071,Y 120.1163,Z 163,A 114.9252,B 19.5994,C -0.6895,E1 19.5387,E2 693.4024} C_DIS
LIN {X -59.0574,Y 121.6447,Z 163,A 113.4753,B 19.5994,C -0.6915,E1 19.5423,E2 694.8513} C_DIS
LIN {X -55.9833,Y 123.0898,Z 163,A 112.0317,B 19.5992,C -0.6934,E1 19.546,E2 696.2938} C_DIS
LIN {X -52.888,Y 124.4511,Z 163,A 110.5954,B 19.5992,C -0.6952,E1 19.5496,E2 697.7291} C_DIS
LIN {X -50.26,Y 125.533,Z 163,A 109.3998,B 19.5992,C -0.6972,E1 19.5527,E2 698.9222} C_DIS
LIN {X -47.1417,Y 126.737,Z 163,A 107.9211,B 19.5992,C -0.6965,E1 19.5566,E2 700.4071} C_DIS
LIN {X -43.5078,Y 128.0324,Z 163,A 106.3311,B 19.599,C -0.7001,E1 19.5608,E2 701.9901} C_DIS
LIN {X -40.3603,Y 129.0591,Z 163,A 104.926,B 19.599,C -0.7016,E1 19.5645,E2 703.3942} C_DIS
LIN {X -37.2077,Y 130.0031,Z 163,A 103.53,B 19.599,C -0.7029,E1 19.5683,E2 704.7892} C_DIS
LIN {X -34.5376,Y 130.7356,Z 163,A 102.3483,B 19.5989,C -0.7037,E1 19.5714,E2 705.9709} C_DIS
LIN {X -31.1799,Y 131.5775,Z 163,A 100.8707,B 19.5989,C -0.7046,E1 19.5755,E2 707.4485} C_DIS
LIN {X -27.749,Y 132.345,Z 163,A 99.3966,B 19.5989,C -0.7064,E1 19.5795,E2 708.9196} C_DIS
LIN {X -23.5058,Y 133.1622,Z 163,A 97.5241,B 19.5989,C -0.7061,E1 19.5846,E2 710.7956} C_DIS
LIN {X -19.9086,Y 133.7493,Z 163,A 96.0205,B 19.5987,C -0.7087,E1 19.5887,E2 712.2934} C_DIS
LIN {X -16.7933,Y 134.176,Z 163,A 94.5291,B 19.5989,C -0.703,E1 19.5929,E2 713.803} C_DIS
LIN {X -13.0731,Y 134.5873,Z 163,A 93.0639,B 19.5987,C -0.7086,E1 19.597,E2 715.2525} C_DIS
LIN {X -9.6952,Y 134.8727,Z 163,A 91.669,B 19.5987,C -0.7108,E1 19.6008,E2 716.6415} C_DIS
LIN {X -6.0283,Y 135.0884,Z 163,A 90.1141,B 19.5987,C -0.7114,E1 19.6052,E2 718.1955} C_DIS
LIN {X -3.0014,Y 135.1895,Z 163,A 88.8323,B 19.5987,C -0.7117,E1 19.6087,E2 719.4764} C_DIS
LIN {X 0.4365,Y 135.2204,Z 163,A 87.3201,B 19.5987,C -0.7097,E1 19.613,E2 720.9946} C_DIS
LIN {X 3.9045,Y 135.1644,Z 163,A 85.8362,B 19.5987,C -0.7092,E1 19.6171,E2 722.4795} C_DIS
LIN {X 6.9385,Y 135.0426,Z 163,A 84.5465,B 19.5987,C -0.7092,E1 19.6207,E2 723.769} C_DIS
LIN {X 10.612,Y 134.8058,Z 163,A 83.0515,B 19.5987,C -0.7116,E1 19.6249,E2 725.2557} C_DIS
LIN {X 14.619,Y 134.4281,Z 163,A 81.3036,B 19.5987,C -0.7096,E1 19.6297,E2 727.008} C_DIS
LIN {X 18.3491,Y 133.9721,Z 163,A 79.7497,B 19.5987,C -0.7107,E1 19.634,E2 728.5569} C_DIS
LIN {X 21.4714,Y 133.5073,Z 163,A 78.4107,B 19.5987,C -0.7102,E1 19.6377,E2 729.8958} C_DIS
LIN {X 24.2392,Y 133.0309,Z 163,A 77.1932,B 19.5987,C -0.7086,E1 19.6411,E2 731.1163} C_DIS
LIN {X 27.749,Y 132.345,Z 163,A 75.7041,B 19.5987,C -0.7089,E1 19.6451,E2 732.602} C_DIS
LIN {X 31.8253,Y 131.422,Z 163,A 73.9301,B 19.5987,C -0.7078,E1 19.65,E2 734.3761} C_DIS
LIN {X 34.9961,Y 130.6134,Z 163,A 72.5309,B 19.5988,C -0.7064,E1 19.6537,E2 735.7766} C_DIS
LIN {X 38.7844,Y 129.5414,Z 163,A 70.8798,B 19.5988,C -0.7058,E1 19.6582,E2 737.4258} C_DIS
LIN {X 41.9349,Y 128.5562,Z 163,A 69.4822,B 19.5988,C -0.7048,E1 19.6619,E2 738.8232} C_DIS
LIN {X 44.5351,Y 127.6762,Z 163,A 68.3067,B 19.5989,C -0.7032,E1 19.665,E2 740.0002} C_DIS
LIN {X 48.2125,Y 126.3359,Z 163,A 66.6643,B 19.5989,C -0.7023,E1 19.6693,E2 741.6409} C_DIS
LIN {X 51.3334,Y 125.1003,Z 163,A 65.2441,B 19.5989,C -0.7009,E1 19.673,E2 743.061} C_DIS
LIN {X 54.4381,Y 123.7809,Z 163,A 63.8176,B 19.599,C -0.6994,E1 19.6766,E2 744.4873} C_DIS
LIN {X 57.5232,Y 122.3777,Z 163,A 62.3845,B 19.599,C -0.6978,E1 19.6803,E2 745.9204} C_DIS
LIN {X 60.5855,Y 120.8909,Z 163,A 60.9456,B 19.5992,C -0.6962,E1 19.6839,E2 747.3592} C_DIS
LIN {X 63.3751,Y 119.4505,Z 163,A 59.703,B 19.5991,C -0.6981,E1 19.6869,E2 748.5913} C_DIS
LIN {X 66.6286,Y 117.6684,Z 163,A 57.9397,B 19.5994,C -0.6878,E1 19.6913,E2 750.3786} C_DIS
LIN {X 70.3407,Y 115.4877,Z 163,A 56.1401,B 19.5994,C -0.6861,E1 19.6956,E2 752.1758} C_DIS
LIN {X 73.9953,Y 113.1809,Z 163,A 54.3265,B 19.5996,C -0.684,E1 19.6998,E2 753.9881} C_DIS
LIN {X 77.586,Y 110.7503,Z 163,A 52.4653,B 19.5997,C -0.6799,E1 19.7041,E2 755.853} C_DIS
LIN {X 81.0852,Y 108.2145,Z 163,A 50.6387,B 19.5998,C -0.6769,E1 19.7082,E2 757.6801} C_DIS
LIN {X 84.5514,Y 105.5285,Z 163,A 48.7916,B 19.5998,C -0.674,E1 19.7123,E2 759.5268} C_DIS
LIN {X 87.9141,Y 102.744,Z 163,A 46.9504,B 19.6,C -0.6708,E1 19.7162,E2 761.3682} C_DIS
LIN {X 91.1892,Y 99.8486,Z 163,A 45.1492,B 19.6,C -0.6693,E1 19.7199,E2 763.1643} C_DIS
LIN {X 94.2661,Y 96.9485,Z 163,A 43.35,B 19.6002,C -0.6653,E1 19.7236,E2 764.9657} C_DIS
LIN {X 97.3797,Y 93.8207,Z 163,A 41.4845,B 19.6003,C -0.6615,E1 19.7272,E2 766.832} C_DIS
LIN {X 100.4363,Y 90.5415,Z 163,A 39.6229,B 19.6003,C -0.6589,E1 19.7307,E2 768.6905} C_DIS
LIN {X 103.3099,Y 87.2484,Z 163,A 37.7685,B 19.6005,C -0.6546,E1 19.7341,E2 770.5467} C_DIS
LIN {X 106.0718,Y 83.8689,Z 163,A 35.9322,B 19.6007,C -0.6508,E1 19.7373,E2 772.383} C_DIS
LIN {X 108.7184,Y 80.4085,Z 163,A 34.0981,B 19.6007,C -0.6468,E1 19.7404,E2 774.2174} C_DIS
LIN {X 111.2462,Y 76.8733,Z 163,A 32.2577,B 19.6009,C -0.6423,E1 19.7434,E2 776.0595} C_DIS
LIN {X 113.6522,Y 73.2692,Z 163,A 30.4169,B 19.6011,C -0.6374,E1 19.7462,E2 777.9027} C_DIS
LIN {X 115.934,Y 69.6026,Z 163,A 28.6315,B 19.6011,C -0.6346,E1 19.7488,E2 779.6846} C_DIS
LIN {X 118.0708,Y 65.9126,Z 163,A 26.8046,B 19.6013,C -0.6289,E1 19.7513,E2 781.5159} C_DIS
LIN {X 120.1163,Y 62.1071,Z 163,A 25.1035,B 19.6013,C -0.6297,E1 19.7535,E2 783.2031} C_DIS
LIN {X 121.6447,Y 59.0574,Z 163,A 23.6698,B 19.6014,C -0.6262,E1 19.7553,E2 784.637} C_DIS
LIN {X 122.8794,Y 56.4382,Z 163,A 22.4189,B 19.6016,C -0.6218,E1 19.7568,E2 785.8922} C_DIS
LIN {X 124.4511,Y 52.888,Z 163,A 20.822,B 19.6016,C -0.6192,E1 19.7585,E2 787.4853} C_DIS
LIN {X 125.7286,Y 49.7748,Z 163,A 19.4083,B 19.6017,C -0.6157,E1 19.76,E2 788.8993} C_DIS
LIN {X 126.7412,Y 47.1305,Z 163,A 18.1862,B 19.6019,C -0.6113,E1 19.7612,E2 790.1255} C_DIS
LIN {X 128.0324,Y 43.5078,Z 163,A 16.6041,B 19.6019,C -0.6086,E1 19.7627,E2 791.7039} C_DIS
LIN {X 129.0591,Y 40.3603,Z 163,A 15.2139,B 19.6021,C -0.605,E1 19.7639,E2 793.0944} C_DIS
LIN {X 129.9676,Y 37.3287,Z 163,A 13.9084,B 19.6021,C -0.6026,E1 19.7649,E2 794.3972} C_DIS
LIN {X 130.7024,Y 34.6622,Z 163,A 12.7077,B 19.6023,C -0.5978,E1 19.7658,E2 795.603} C_DIS
LIN {X 131.6452,Y 30.8991,Z 163,A 11.0957,B 19.6023,C -0.5943,E1 19.7668,E2 797.2134} C_DIS
LIN {X 132.2898,Y 28.0047,Z 163,A 9.8451,B 19.6025,C -0.5907,E1 19.7676,E2 798.465} C_DIS
LIN {X 132.905,Y 24.9212,Z 163,A 8.512,B 19.6025,C -0.5866,E1 19.7683,E2 799.8001} C_DIS
LIN {X 133.652,Y 20.537,Z 163,A 6.6894,B 19.6027,C -0.5836,E1 19.7691,E2 801.6177} C_DIS
LIN {X 134.094,Y 17.4188,Z 163,A 5.3122,B 19.6029,C -0.5775,E1 19.7696,E2 803.0021} C_DIS
LIN {X 134.5277,Y 13.6936,Z 163,A 3.7711,B 19.6029,C -0.5747,E1 19.7701,E2 804.5397} C_DIS
LIN {X 134.8058,Y 10.612,Z 163,A 2.4735,B 19.603,C -0.5712,E1 19.7704,E2 805.8375} C_DIS
LIN {X 135.0884,Y 6.0283,Z 163,A 0.3853,B 19.6034,C -0.5588,E1 19.7707,E2 807.9464} C_DIS
LIN {X 135.2032,Y 2.1802,Z 163,A -1.111,B 19.6034,C -0.5597,E1 19.7708,E2 809.4283} C_DIS
LIN {X 135.2146,Y -1.4974,Z 163,A -2.6137,B 19.6034,C -0.5572,E1 19.7708,E2 810.9266} C_DIS
LIN {X 135.1644,Y -3.9045,Z 163,A -3.6933,B 19.6036,C -0.5514,E1 19.7708,E2 812.0151} C_DIS
LIN {X 134.974,Y -8.165,Z 163,A -5.4624,B 19.6036,C -0.5474,E1 19.7705,E2 813.7823} C_DIS
LIN {X 134.7219,Y -11.6055,Z 163,A -6.9294,B 19.6038,C -0.5426,E1 19.7701,E2 815.2522} C_DIS
LIN {X 134.3612,Y -15.2413,Z 163,A -8.4136,B 19.6038,C -0.5405,E1 19.7697,E2 816.731} C_DIS
LIN {X 133.9721,Y -18.3491,Z 163,A -9.7315,B 19.604,C -0.5367,E1 19.7692,E2 818.0498} C_DIS
LIN {X 133.246,Y -23.0371,Z 163,A -11.7288,B 19.6041,C -0.531,E1 19.7683,E2 820.0488} C_DIS
LIN {X 132.6651,Y -26.1763,Z 163,A -13.0726,B 19.6042,C -0.5272,E1 19.7676,E2 821.3937} C_DIS
LIN {X 132.0051,Y -29.3234,Z 163,A -14.426,B 19.6043,C -0.5234,E1 19.7668,E2 822.7481} C_DIS
LIN {X 131.2652,Y -32.4757,Z 163,A -15.7889,B 19.6044,C -0.5195,E1 19.766,E2 824.112} C_DIS
LIN {X 130.4442,Y -35.6304,Z 163,A -17.1613,B 19.6045,C -0.5156,E1 19.765,E2 825.4856} C_DIS
LIN {X 129.5414,Y -38.7844,Z 163,A -18.5418,B 19.6046,C -0.5118,E1 19.7639,E2 826.8671} C_DIS
LIN {X 128.5562,Y -41.9349,Z 163,A -19.9311,B 19.6047,C -0.5079,E1 19.7627,E2 828.2576} C_DIS
LIN {X 127.6372,Y -44.6476,Z 163,A -21.1737,B 19.6048,C -0.503,E1 19.7616,E2 829.5056} C_DIS
LIN {X 126.3359,Y -48.2125,Z 163,A -22.7336,B 19.6048,C -0.5003,E1 19.7601,E2 831.0622} C_DIS
LIN {X 125.1003,Y -51.3334,Z 163,A -24.1465,B 19.605,C -0.4964,E1 19.7586,E2 832.4763} C_DIS
LIN {X 123.7809,Y -54.4381,Z 163,A -25.5661,B 19.605,C -0.4927,E1 19.757,E2 833.8969} C_DIS
LIN {X 122.3777,Y -57.5232,Z 163,A -26.9926,B 19.6052,C -0.4889,E1 19.7553,E2 835.3246} C_DIS
LIN {X 120.9591,Y -60.4474,Z 163,A -28.3654,B 19.6052,C -0.4851,E1 19.7536,E2 836.699} C_DIS
LIN {X 119.3209,Y -63.6218,Z 163,A -29.8235,B 19.6053,C -0.4832,E1 19.7518,E2 838.1526} C_DIS
LIN {X 117.7388,Y -66.5033,Z 163,A -31.3176,B 19.6055,C -0.4747,E1 19.7497,E2 839.6615} C_DIS
LIN {X 115.4877,Y -70.3407,Z 163,A -33.2318,B 19.6057,C -0.4682,E1 19.747,E2 841.5823} C_DIS
LIN {X 113.1809,Y -73.9953,Z 163,A -35.0209,B 19.6057,C -0.465,E1 19.7443,E2 843.369} C_DIS
LIN {X 110.7503,Y -77.586,Z 163,A -36.8728,B 19.6059,C -0.4594,E1 19.7413,E2 845.2256} C_DIS
LIN {X 108.1985,Y -81.1068,Z 163,A -38.7076,B 19.6059,C -0.4549,E1 19.7383,E2 847.0622} C_DIS
LIN {X 105.5285,Y -84.5514,Z 163,A -40.5427,B 19.6061,C -0.4506,E1 19.7351,E2 848.8987} C_DIS
LIN {X 102.744,Y -87.9141,Z 163,A -42.381,B 19.6061,C -0.4465,E1 19.7318,E2 850.7383} C_DIS
LIN {X 99.8486,Y -91.1892,Z 163,A -44.2217,B 19.6062,C -0.4424,E1 19.7283,E2 852.5803} C_DIS
LIN {X 96.8466,Y -94.3713,Z 163,A -46.0328,B 19.6062,C -0.4398,E1 19.7249,E2 854.3888} C_DIS
LIN {X 93.7426,Y -97.4553,Z 163,A -47.8754,B 19.6064,C -0.436,E1 19.7212,E2 856.2326} C_DIS
LIN {X 90.5415,Y -100.4363,Z 163,A -49.7052,B 19.6064,C -0.4329,E1 19.7174,E2 858.0621} C_DIS
LIN {X 87.2484,Y -103.3099,Z 163,A -51.5584,B 19.6065,C -0.4288,E1 19.7135,E2 859.918} C_DIS
LIN {X 83.8689,Y -106.0718,Z 163,A -53.4275,B 19.6066,C -0.424,E1 19.7094,E2 861.792} C_DIS
LIN {X 80.4595,Y -108.6804,Z 163,A -55.212,B 19.6066,C -0.4218,E1 19.7054,E2 863.5747} C_DIS
LIN {X 76.8733,Y -111.2462,Z 163,A -57.0932,B 19.6068,C -0.4175,E1 19.7011,E2 865.4599} C_DIS
LIN {X 73.2692,Y -113.6522,Z 163,A -58.9188,B 19.6068,C -0.4146,E1 19.6968,E2 867.2865} C_DIS
LIN {X 69.6026,Y -115.934,Z 163,A -60.7081,B 19.6068,C -0.413,E1 19.6926,E2 869.0729} C_DIS
LIN {X 65.8798,Y -118.0892,Z 163,A -62.5511,B 19.6069,C -0.409,E1 19.6881,E2 870.9206} C_DIS
LIN {X 62.1071,Y -120.1163,Z 163,A -64.2455,B 19.6069,C -0.4112,E1 19.684,E2 872.6022} C_DIS
LIN {X 59.0574,Y -121.6447,Z 163,A -65.6836,B 19.6069,C -0.4093,E1 19.6804,E2 874.041} C_DIS
LIN {X 56.3546,Y -122.9181,Z 163,A -66.9731,B 19.6069,C -0.4064,E1 19.6771,E2 875.3347} C_DIS
LIN {X 52.888,Y -124.4511,Z 163,A -68.5417,B 19.6069,C -0.4057,E1 19.6731,E2 876.9004} C_DIS
LIN {X 49.7748,Y -125.7286,Z 163,A -69.9611,B 19.607,C -0.4041,E1 19.6694,E2 878.3205} C_DIS
LIN {X 46.647,Y -126.9223,Z 163,A -71.373,B 19.607,C -0.4025,E1 19.6657,E2 879.733} C_DIS
LIN {X 43.9988,Y -127.8621,Z 163,A -72.6045,B 19.6071,C -0.3994,E1 19.6624,E2 880.9707} C_DIS
LIN {X 40.3603,Y -129.0591,Z 163,A -74.1744,B 19.6071,C -0.3998,E1 19.6583,E2 882.5355} C_DIS
LIN {X 37.2077,Y -130.0031,Z 163,A -75.5627,B 19.6071,C -0.3985,E1 19.6545,E2 883.9244} C_DIS
LIN {X 34.053,Y -130.8649,Z 163,A -76.9433,B 19.6071,C -0.3974,E1 19.6508,E2 885.3056} C_DIS
LIN {X 29.3234,Y -132.0051,Z 163,A -78.9963,B 19.6071,C -0.3959,E1 19.6452,E2 887.3592} C_DIS
LIN {X 26.1763,Y -132.6651,Z 163,A -80.3539,B 19.6072,C -0.395,E1 19.6415,E2 888.7174} C_DIS
LIN {X 23.2628,Y -133.2056,Z 163,A -81.5909,B 19.6072,C -0.3948,E1 19.6381,E2 889.9529} C_DIS
LIN {X 19.9086,Y -133.7493,Z 163,A -83.04,B 19.6072,C -0.3934,E1 19.6341,E2 891.4043} C_DIS
LIN {X 15.8653,Y -134.2867,Z 163,A -84.7044,B 19.6072,C -0.3952,E1 19.6295,E2 893.0618} C_DIS
LIN {X 13.0731,Y -134.5873,Z 163,A -85.9482,B 19.6072,C -0.3923,E1 19.6261,E2 894.3131} C_DIS
LIN {X 9.7859,Y -134.8661,Z 163,A -87.3566,B 19.6072,C -0.3912,E1 19.6221,E2 895.7237} C_DIS
LIN {X 6.0283,Y -135.0884,Z 163,A -88.9324,B 19.6072,C -0.3914,E1 19.6177,E2 897.2981} C_DIS
LIN {X 3.0014,Y -135.1895,Z 163,A -90.2126,B 19.6072,C -0.3912,E1 19.6142,E2 898.5787} C_DIS
LIN {X 3.0014,Y -135.1895,Z 163,A -90.2126,B 19.6072,C -0.3912,E1 19.6142,E2 898.5787} C_DIS
Enddeposition()
LIN {X 0.9453,Y -134.2958,Z 163,A -90.5739,B 18.3821,C -0.2588,E1 18.3851,E2 899.2524} C_DIS
Startdeposition()
$VEL.CP = VEL_PRINT
LIN {X 3.4297,Y -134.2564,Z 163,A -89.0437,B 18.3818,C -0.2775,E1 18.3895,E2 897.6634} C_DIS
LIN {X 7.2906,Y -134.1029,Z 163,A -87.2878,B 18.3818,C -0.2823,E1 18.3944,E2 895.8932} C_DIS
LIN {X 11.2706,Y -133.826,Z 163,A -85.7025,B 18.3818,C -0.2784,E1 18.3988,E2 894.3214} C_DIS
LIN {X 15.3278,Y -133.4234,Z 163,A -83.8906,B 18.3818,C -0.2821,E1 18.4039,E2 892.4994} C_DIS
LIN {X 19.072,Y -132.9385,Z 163,A -82.3681,B 18.3818,C -0.2796,E1 18.408,E2 890.9867} C_DIS
LIN {X 22.8012,Y -132.3518,Z 163,A -80.6442,B 18.3818,C -0.2852,E1 18.4128,E2 889.2475} C_DIS
LIN {X 26.5458,Y -131.6501,Z 163,A -79.0763,B 18.3818,C -0.2842,E1 18.4171,E2 887.6855} C_DIS
LIN {X 30.6789,Y -130.7509,Z 163,A -77.2073,B 18.3817,C -0.2883,E1 18.4222,E2 885.8071} C_DIS
LIN {X 34.9847,Y -129.6633,Z 163,A -75.0986,B 18.3815,C -0.2988,E1 18.428,E2 883.6698} C_DIS
LIN {X 38.4785,Y -128.6714,Z 163,A -73.4376,B 18.3814,C -0.3049,E1 18.4325,E2 881.9935} C_DIS
LIN {X 42.2744,Y -127.4724,Z 163,A -72.2048,B 18.3817,C -0.288,E1 18.4356,E2 880.8175} C_DIS
LIN {X 45.5069,Y -126.3544,Z 163,A -70.7446,B 18.3817,C -0.2898,E1 18.4395,E2 879.3558} C_DIS
LIN {X 48.4159,Y -125.2688,Z 163,A -69.3564,B 18.3816,C -0.2941,E1 18.4431,E2 877.9584} C_DIS
LIN {X 51.8312,Y -123.8944,Z 163,A -67.9194,B 18.3816,C -0.2908,E1 18.4468,E2 876.5365} C_DIS
LIN {X 54.4922,Y -122.7479,Z 163,A -66.6034,B 18.3816,C -0.2958,E1 18.4502,E2 875.2092} C_DIS
LIN {X 57.1258,Y -121.5469,Z 163,A -65.3776,B 18.3816,C -0.2972,E1 18.4533,E2 873.9833} C_DIS
LIN {X 60.3879,Y -119.9581,Z 163,A -63.7888,B 18.3815,C -0.3013,E1 18.4573,E2 872.3876} C_DIS
LIN {X 63.9414,Y -118.1036,Z 163,A -62.1188,B 18.3815,C -0.3024,E1 18.4614,E2 870.7208} C_DIS
LIN {X 67.794,Y -115.9348,Z 163,A -60.1959,B 18.3814,C -0.3071,E1 18.466,E2 868.7911} C_DIS
LIN {X 72.2111,Y -113.2362,Z 163,A -57.9928,B 18.3814,C -0.3108,E1 18.4713,E2 866.586} C_DIS
LIN {X 75.7288,Y -110.9147,Z 163,A -56.172,B 18.3812,C -0.3152,E1 18.4755,E2 864.7602} C_DIS
LIN {X 79.478,Y -108.2593,Z 163,A -54.4025,B 18.3812,C -0.3111,E1 18.4795,E2 863.0121} C_DIS
LIN {X 82.3852,Y -106.0638,Z 163,A -52.7199,B 18.3812,C -0.3196,E1 18.4832,E2 861.3114} C_DIS
LIN {X 85.9048,Y -103.2341,Z 163,A -50.8214,B 18.3812,C -0.3225,E1 18.4873,E2 859.4139} C_DIS
LIN {X 89.0225,Y -100.5576,Z 163,A -49.0673,B 18.381,C -0.3264,E1 18.491,E2 857.6573} C_DIS
LIN {X 91.8938,Y -97.9412,Z 163,A -47.4972,B 18.381,C -0.3264,E1 18.4942,E2 856.096} C_DIS
LIN {X 94.7201,Y -95.2099,Z 163,A -45.7753,B 18.381,C -0.3322,E1 18.4977,E2 854.3661} C_DIS
LIN {X 97.5679,Y -92.2895,Z 163,A -44.0255,B 18.3809,C -0.3367,E1 18.5011,E2 852.6127} C_DIS
LIN {X 100.4111,Y -89.1881,Z 163,A -42.3809,B 18.3809,C -0.3348,E1 18.5041,E2 850.9844} C_DIS
LIN {X 102.526,Y -86.7487,Z 163,A -40.617,B 18.3805,C -0.3544,E1 18.5074,E2 849.17} C_DIS
LIN {X 104.7385,Y -84.064,Z 163,A -39.3693,B 18.3807,C -0.3482,E1 18.5096,E2 847.9499} C_DIS
LIN {X 107.3958,Y -80.6416,Z 163,A -37.5414,B 18.3806,C -0.3521,E1 18.5126,E2 846.1218} C_DIS
LIN {X 110.0109,Y -77.0363,Z 163,A -35.6298,B 18.3805,C -0.3576,E1 18.5157,E2 844.2061} C_DIS
LIN {X 112.2783,Y -73.6916,Z 163,A -33.6608,B 18.3802,C -0.3725,E1 18.5188,E2 842.2036} C_DIS
LIN {X 114.3,Y -70.5156,Z 163,A -32.3285,B 18.3803,C -0.3654,E1 18.5207,E2 840.9034} C_DIS
LIN {X 116.5452,Y -66.739,Z 163,A -30.3781,B 18.3802,C -0.3738,E1 18.5235,E2 838.9406} C_DIS
LIN {X 118.7606,Y -62.708,Z 163,A -28.6911,B 18.3802,C -0.3677,E1 18.5257,E2 837.285} C_DIS
LIN {X 119.993,Y -60.3195,Z 163,A -27.4121,B 18.3802,C -0.3766,E1 18.5273,E2 835.9878} C_DIS
LIN {X 121.7609,Y -56.6628,Z 163,A -25.7696,B 18.3801,C -0.3778,E1 18.5293,E2 834.3539} C_DIS
LIN {X 123.2081,Y -53.4423,Z 163,A -24.466,B 18.3801,C -0.3736,E1 18.5307,E2 833.0733} C_DIS
LIN {X 124.4732,Y -50.426,Z 163,A -22.9802,B 18.3801,C -0.3815,E1 18.5323,E2 831.5741} C_DIS
LIN {X 125.5083,Y -47.7966,Z 163,A -21.591,B 18.3798,C -0.3928,E1 18.5338,E2 830.1601} C_DIS
LIN {X 126.8316,Y -44.1599,Z 163,A -20.0779,B 18.3798,C -0.3919,E1 18.5352,E2 828.6617} C_DIS
LIN {X 127.7485,Y -41.4368,Z 163,A -18.7743,B 18.3797,C -0.3989,E1 18.5363,E2 827.3465} C_DIS
LIN {X 128.9441,Y -37.5473,Z 163,A -17.137,B 18.3797,C -0.4,E1 18.5376,E2 825.7188} C_DIS
LIN {X 130.0358,Y -33.5759,Z 163,A -15.365,B 18.3795,C -0.406,E1 18.5389,E2 823.9423} C_DIS
LIN {X 130.7535,Y -30.667,Z 163,A -14.0495,B 18.3794,C -0.4115,E1 18.5397,E2 822.6202} C_DIS
LIN {X 131.7975,Y -25.8094,Z 163,A -11.971,B 18.3793,C -0.4162,E1 18.5409,E2 820.5437} C_DIS
LIN {X 132.4937,Y -21.9503,Z 163,A -10.3439,B 18.3793,C -0.4195,E1 18.5417,E2 818.9197} C_DIS
LIN {X 133.0635,Y -18.1951,Z 163,A -8.6631,B 18.3791,C -0.427,E1 18.5424,E2 817.229} C_DIS
LIN {X 133.5189,Y -14.4611,Z 163,A -7.1153,B 18.379,C -0.4297,E1 18.5428,E2 815.6858} C_DIS
LIN {X 133.916,Y -10.1525,Z 163,A -5.2832,B 18.3789,C -0.4348,E1 18.5433,E2 813.8528} C_DIS
LIN {X 134.1577,Y -6.1997,Z 163,A -3.6152,B 18.3788,C -0.4392,E1 18.5435,E2 812.1849} C_DIS
LIN {X 134.2798,Y -2.3223,Z 163,A -1.9983,B 18.3787,C -0.4427,E1 18.5436,E2 810.5704} C_DIS
LIN {X 134.2861,Y 1.9411,Z 163,A -0.1639,B 18.3785,C -0.449,E1 18.5436,E2 808.7314} C_DIS
LIN {X 134.1588,Y 6.1787,Z 163,A 1.6243,B 18.3785,C -0.4538,E1 18.5434,E2 806.9432} C_DIS
LIN {X 133.9456,Y 9.7461,Z 163,A 3.1153,B 18.3784,C -0.4571,E1 18.5431,E2 805.4541} C_DIS
LIN {X 133.5658,Y 14.0247,Z 163,A 4.941,B 18.3782,C -0.4624,E1 18.5426,E2 803.6267} C_DIS
LIN {X 133.1357,Y 17.6444,Z 163,A 6.5021,B 18.3782,C -0.4674,E1 18.5421,E2 802.0627} C_DIS
LIN {X 132.4732,Y 22.0736,Z 163,A 8.3063,B 18.3781,C -0.4688,E1 18.5413,E2 800.2692} C_DIS
LIN {X 131.8863,Y 25.3453,Z 163,A 9.7958,B 18.3779,C -0.4761,E1 18.5405,E2 798.7689} C_DIS
LIN {X 130.8294,Y 30.335,Z 163,A 11.8961,B 18.3779,C -0.4794,E1 18.5393,E2 796.6752} C_DIS
LIN {X 129.8523,Y 34.2759,Z 163,A 13.5933,B 18.3777,C -0.4831,E1 18.5381,E2 794.98} C_DIS
LIN {X 128.9588,Y 37.497,Z 163,A 15.0614,B 18.3776,C -0.4891,E1 18.537,E2 793.5049} C_DIS
LIN {X 127.9359,Y 40.8502,Z 163,A 16.5211,B 18.3775,C -0.492,E1 18.5358,E2 792.0477} C_DIS
LIN {X 126.5127,Y 45.0679,Z 163,A 18.4578,B 18.3773,C -0.499,E1 18.534,E2 790.1041} C_DIS
LIN {X 125.2638,Y 48.429,Z 163,A 19.9242,B 18.3773,C -0.5007,E1 18.5326,E2 788.6438} C_DIS
LIN {X 124.0657,Y 51.4213,Z 163,A 21.2945,B 18.3772,C -0.5044,E1 18.5311,E2 787.2725} C_DIS
LIN {X 122.6615,Y 54.6854,Z 163,A 22.7697,B 18.3771,C -0.507,E1 18.5295,E2 785.8005} C_DIS
LIN {X 121.1961,Y 57.8601,Z 163,A 25.1905,B 18.3759,C -0.55,E1 18.5264,E2 783.2623} C_DIS
LIN {X 118.15,Y 63.8554,Z 163,A 27.1293,B 18.3768,C -0.5187,E1 18.524,E2 781.4367} C_DIS
LIN {X 115.9125,Y 67.8318,Z 163,A 29.1336,B 18.3766,C -0.5262,E1 18.5212,E2 779.4233} C_DIS
LIN {X 113.6982,Y 71.4815,Z 163,A 30.9622,B 18.3764,C -0.5312,E1 18.5185,E2 777.5919} C_DIS
LIN {X 111.4615,Y 74.9222,Z 163,A 32.7053,B 18.3764,C -0.5352,E1 18.5158,E2 775.8481} C_DIS
LIN {X 108.9181,Y 78.5732,Z 163,A 34.6014,B 18.3762,C -0.5398,E1 18.5128,E2 773.9506} C_DIS
LIN {X 106.1396,Y 82.2873,Z 163,A 36.5004,B 18.3762,C -0.5413,E1 18.5096,E2 772.0597} C_DIS
LIN {X 103.5108,Y 85.5708,Z 163,A 38.3257,B 18.376,C -0.5467,E1 18.5063,E2 770.2291} C_DIS
LIN {X 100.4917,Y 89.097,Z 163,A 40.2621,B 18.376,C -0.5493,E1 18.5028,E2 768.2967} C_DIS
LIN {X 97.5094,Y 92.3515,Z 163,A 42.1608,B 18.3758,C -0.5541,E1 18.4992,E2 766.3947} C_DIS
LIN {X 94.3836,Y 95.5442,Z 163,A 44.0768,B 18.3756,C -0.5585,E1 18.4954,E2 764.4762} C_DIS
LIN {X 91.2487,Y 98.5425,Z 163,A 45.905,B 18.3756,C -0.5613,E1 18.4917,E2 762.6496} C_DIS
LIN {X 87.8998,Y 101.5409,Z 163,A 47.8169,B 18.3755,C -0.5648,E1 18.4877,E2 760.7373} C_DIS
LIN {X 84.5555,Y 104.3422,Z 163,A 49.6433,B 18.3754,C -0.5669,E1 18.4837,E2 758.9142} C_DIS
LIN {X 81.1477,Y 107.0139,Z 163,A 51.4963,B 18.3753,C -0.5704,E1 18.4796,E2 757.0595} C_DIS
LIN {X 77.6244,Y 109.5963,Z 163,A 53.3682,B 18.3752,C -0.5739,E1 18.4754,E2 755.1858} C_DIS
LIN {X 73.756,Y 112.2359,Z 163,A 55.3263,B 18.3752,C -0.5756,E1 18.4708,E2 753.2317} C_DIS
LIN {X 69.9017,Y 114.6766,Z 163,A 58.1751,B 18.3739,C -0.615,E1 18.4638,E2 750.2707} C_DIS
LIN {X 63.8493,Y 118.1533,Z 163,A 60.5614,B 18.3745,C -0.5952,E1 18.4581,E2 747.9571} C_DIS
LIN {X 60.4651,Y 119.9188,Z 163,A 61.8899,B 18.3748,C -0.5852,E1 18.4549,E2 746.6649} C_DIS
LIN {X 56.4977,Y 121.8373,Z 163,A 63.6438,B 18.3749,C -0.5825,E1 18.4505,E2 744.9261} C_DIS
LIN {X 53.2866,Y 123.2755,Z 163,A 65.1163,B 18.3749,C -0.5831,E1 18.4468,E2 743.4569} C_DIS
LIN {X 50.5622,Y 124.4183,Z 163,A 66.2752,B 18.3749,C -0.5804,E1 18.4438,E2 742.3103} C_DIS
LIN {X 47.3113,Y 125.6901,Z 163,A 67.9058,B 18.3748,C -0.5874,E1 18.4395,E2 740.6623} C_DIS
LIN {X 44.0713,Y 126.8623,Z 163,A 69.1309,B 18.375,C -0.5792,E1 18.4364,E2 739.467} C_DIS
LIN {X 41.3357,Y 127.7808,Z 163,A 70.6529,B 18.3746,C -0.5916,E1 18.4322,E2 737.9096} C_DIS
LIN {X 37.5682,Y 128.938,Z 163,A 72.3208,B 18.3746,C -0.5924,E1 18.4278,E2 736.2434} C_DIS
LIN {X 33.3562,Y 130.0916,Z 163,A 73.9141,B 18.3749,C -0.5831,E1 18.4236,E2 734.6831} C_DIS
LIN {X 29.0399,Y 131.1242,Z 163,A 76.1207,B 18.3745,C -0.5964,E1 18.4175,E2 732.4388} C_DIS
LIN {X 25.3581,Y 131.8839,Z 163,A 77.6049,B 18.3746,C -0.5925,E1 18.4134,E2 730.9694} C_DIS
LIN {X 21.7635,Y 132.5249,Z 163,A 79.2546,B 18.3745,C -0.5967,E1 18.4089,E2 729.3089} C_DIS
LIN {X 17.5142,Y 133.1527,Z 163,A 80.9784,B 18.3746,C -0.593,E1 18.4041,E2 727.5988} C_DIS
LIN {X 14.1269,Y 133.5548,Z 163,A 82.5298,B 18.3745,C -0.597,E1 18.3998,E2 726.0362} C_DIS
LIN {X 10.2888,Y 133.906,Z 163,A 84.1658,B 18.3745,C -0.597,E1 18.3952,E2 724.4019} C_DIS
LIN {X 6.582,Y 134.1385,Z 163,A 85.6839,B 18.3745,C -0.5944,E1 18.391,E2 722.8924} C_DIS
LIN {X 2.481,Y 134.2771,Z 163,A 87.4666,B 18.3745,C -0.5956,E1 18.3861,E2 721.1066} C_DIS
LIN {X -1.712,Y 134.2899,Z 163,A 89.3105,B 18.3745,C -0.5974,E1 18.3809,E2 719.2569} C_DIS
LIN {X -5.6943,Y 134.1798,Z 163,A 90.9433,B 18.3745,C -0.5945,E1 18.3764,E2 717.6331} C_DIS
LIN {X -9.7758,Y 133.9435,Z 163,A 92.654,B 18.3746,C -0.5926,E1 18.3716,E2 715.9275} C_DIS
LIN {X -13.5842,Y 133.6131,Z 163,A 94.4178,B 18.3745,C -0.597,E1 18.3667,E2 714.1487} C_DIS
LIN {X -17.4544,Y 133.1606,Z 163,A 95.9959,B 18.3746,C -0.5929,E1 18.3623,E2 712.5818} C_DIS
LIN {X -21.7728,Y 132.5234,Z 163,A 97.8517,B 18.3746,C -0.5916,E1 18.3572,E2 710.7281} C_DIS
LIN {X -25.2392,Y 131.9066,Z 163,A 99.186,B 18.3749,C -0.5842,E1 18.3536,E2 709.4152} C_DIS
LIN {X -28.721,Y 131.1931,Z 163,A 100.945,B 18.3746,C -0.5922,E1 18.3487,E2 707.628} C_DIS
LIN {X -32.6835,Y 130.2623,Z 163,A 102.6219,B 18.3747,C -0.5884,E1 18.3442,E2 705.9598} C_DIS
LIN {X -36.226,Y 129.3214,Z 163,A 104.127,B 18.3749,C -0.5848,E1 18.3402,E2 704.4631} C_DIS
LIN {X -39.9315,Y 128.2273,Z 163,A 106.1129,B 18.3745,C -0.5957,E1 18.3347,E2 702.4378} C_DIS
LIN {X -43.0827,Y 127.2033,Z 163,A 107.3306,B 18.3748,C -0.5868,E1 18.3316,E2 701.2451} C_DIS
LIN {X -46.788,Y 125.8861,Z 163,A 108.9027,B 18.375,C -0.5809,E1 18.3275,E2 699.6874} C_DIS
LIN {X -49.9433,Y 124.6678,Z 163,A 110.3859,B 18.375,C -0.5806,E1 18.3236,E2 698.2007} C_DIS
LIN {X -53.4689,Y 123.1966,Z 163,A 111.995,B 18.375,C -0.5776,E1 18.3195,E2 696.5958} C_DIS
LIN {X -56.878,Y 121.6614,Z 163,A 113.5376,B 18.3752,C -0.5734,E1 18.3156,E2 695.0612} C_DIS
LIN {X -62.7063,Y 118.7615,Z 163,A 116.4102,B 18.3752,C -0.5727,E1 18.3084,E2 692.1802} C_DIS
LIN {X -66.4898,Y 116.6873,Z 163,A 118.334,B 18.3752,C -0.5727,E1 18.3037,E2 690.2486} C_DIS
LIN {X -70.3869,Y 114.3789,Z 163,A 120.193,B 18.3754,C -0.5667,E1 18.2993,E2 688.4006} C_DIS
LIN {X -72.8068,Y 112.8545,Z 163,A 121.569,B 18.3754,C -0.5702,E1 18.296,E2 687.0073} C_DIS
LIN {X -77.4026,Y 109.7527,Z 163,A 123.8722,B 18.3754,C -0.5635,E1 18.2908,E2 684.7145} C_DIS
LIN {X -81.1666,Y 106.9996,Z 163,A 125.6932,B 18.3758,C -0.5535,E1 18.2867,E2 682.9164} C_DIS
LIN {X -85.8274,Y 103.2982,Z 163,A 128.9268,B 18.3752,C -0.5735,E1 18.2796,E2 679.602} C_DIS
LIN {X -89.4594,Y 100.1692,Z 163,A 130.5054,B 18.3758,C -0.5521,E1 18.2764,E2 678.0827} C_DIS
LIN {X -95.4964,Y 94.4318,Z 163,A 133.8145,B 18.3763,C -0.5353,E1 18.2698,E2 674.8081} C_DIS
LIN {X -98.8413,Y 90.9243,Z 163,A 136.3242,B 18.376,C -0.5463,E1 18.2649,E2 672.2479} C_DIS
LIN {X -101.2664,Y 88.2154,Z 163,A 138.6435,B 18.3753,C -0.5703,E1 18.2606,E2 669.8371} C_DIS
LIN {X -105.784,Y 82.7444,Z 163,A 140.7392,B 18.3765,C -0.529,E1 18.2571,E2 667.8595} C_DIS
LIN {X -108.4787,Y 79.1793,Z 163,A 142.6865,B 18.3765,C -0.5256,E1 18.2538,E2 665.91} C_DIS
LIN {X -111.072,Y 75.4976,Z 163,A 144.6261,B 18.3767,C -0.5212,E1 18.2507,E2 663.971} C_DIS
LIN {X -113.5367,Y 71.7374,Z 163,A 146.3325,B 18.377,C -0.5085,E1 18.2482,E2 662.293} C_DIS
LIN {X -115.4097,Y 68.6836,Z 163,A 148.0925,B 18.377,C -0.5125,E1 18.2456,E2 660.5073} C_DIS
LIN {X -117.7023,Y 64.6774,Z 163,A 150.1042,B 18.377,C -0.5086,E1 18.2429,E2 658.4935} C_DIS
LIN {X -119.3869,Y 61.51,Z 163,A 152.042,B 18.3768,C -0.5188,E1 18.2403,E2 656.5085} C_DIS
LIN {X -121.3191,Y 57.6026,Z 163,A 153.4355,B 18.3774,C -0.4969,E1 18.2387,E2 655.1744} C_DIS
LIN {X -123.1138,Y 53.6604,Z 163,A 155.7817,B 18.377,C -0.5092,E1 18.236,E2 652.7705} C_DIS
LIN {X -124.8628,Y 49.4595,Z 163,A 157.3345,B 18.3775,C -0.4897,E1 18.2344,E2 651.268} C_DIS
LIN {X -126.1571,Y 46.0542,Z 163,A 158.8326,B 18.3777,C -0.4831,E1 18.233,E2 649.7791} C_DIS
LIN {X -127.2912,Y 42.8187,Z 163,A 160.0875,B 18.378,C -0.4714,E1 18.2319,E2 648.5515} C_DIS
LIN {X -129.7469,Y 34.6713,Z 163,A 163.9926,B 18.378,C -0.47,E1 18.2288,E2 644.6191} C_DIS
LIN {X -130.645,Y 31.1186,Z 163,A 165.5497,B 18.3782,C -0.4651,E1 18.2277,E2 643.0651} C_DIS
LIN {X -131.5556,Y 27.0101,Z 163,A 167.3186,B 18.3783,C -0.4586,E1 18.2267,E2 641.3021} C_DIS
LIN {X -132.2434,Y 23.4119,Z 163,A 169.0075,B 18.3783,C -0.4583,E1 18.2259,E2 639.6004} C_DIS
LIN {X -132.942,Y 19.0475,Z 163,A 170.7993,B 18.3785,C -0.4491,E1 18.2251,E2 637.8228} C_DIS
LIN {X -133.4372,Y 15.2123,Z 163,A 172.5783,B 18.3785,C -0.4485,E1 18.2245,E2 636.0306} C_DIS
LIN {X -133.7753,Y 11.8702,Z 163,A 174.0322,B 18.3786,C -0.4448,E1 18.2241,E2 634.5763} C_DIS
LIN {X -134.0968,Y 7.4106,Z 163,A 175.7516,B 18.3789,C -0.4322,E1 18.2238,E2 632.8826} C_DIS
LIN {X -134.2304,Y 4.3644,Z 163,A 177.2277,B 18.3789,C -0.4344,E1 18.2237,E2 631.3872} C_DIS
LIN {X -134.3007,Y 0.427,Z 163,A 178.9722,B 18.3789,C -0.4314,E1 18.2237,E2 629.6373} C_DIS
LIN {X -134.2465,Y -3.7852,Z 163,A -179.348,B 18.3792,C -0.4217,E1 18.2237,E2 627.9742} C_DIS
LIN {X -134.0672,Y -7.9084,Z 163,A -177.5206,B 18.3792,C -0.4186,E1 18.224,E2 626.1413} C_DIS
LIN {X -133.7543,Y -12.1075,Z 163,A -175.5257,B 18.3792,C -0.4201,E1 18.2245,E2 624.1248} C_DIS
LIN {X -133.1882,Y -17.244,Z 163,A -173.6069,B 18.3796,C -0.4033,E1 18.2251,E2 622.2438} C_DIS
LIN {X -132.7493,Y -20.348,Z 163,A -172.2167,B 18.3796,C -0.401,E1 18.2257,E2 620.849} C_DIS
LIN {X -131.7667,Y -25.9702,Z 163,A -169.1849,B 18.3793,C -0.4149,E1 18.2273,E2 617.7476} C_DIS
LIN {X -130.814,Y -30.4026,Z 163,A -167.505,B 18.3796,C -0.4,E1 18.2283,E2 616.1014} C_DIS
LIN {X -129.6933,Y -34.8721,Z 163,A -165.7753,B 18.3799,C -0.3858,E1 18.2295,E2 614.4031} C_DIS
LIN {X -128.538,Y -38.9163,Z 163,A -163.942,B 18.38,C -0.3819,E1 18.2309,E2 612.5673} C_DIS
LIN {X -127.3936,Y -42.5113,Z 163,A -162.336,B 18.3801,C -0.3771,E1 18.2323,E2 610.9637} C_DIS
LIN {X -125.9187,Y -46.7011,Z 163,A -160.467,B 18.3802,C -0.3708,E1 18.2341,E2 609.1002} C_DIS
LIN {X -124.7879,Y -49.6453,Z 163,A -159.0853,B 18.3802,C -0.3682,E1 18.2355,E2 607.7157} C_DIS
LIN {X -123.3695,Y -53.069,Z 163,A -157.4846,B 18.3804,C -0.3645,E1 18.2372,E2 606.1143} C_DIS
LIN {X -122.1096,Y -55.9088,Z 163,A -156.1393,B 18.3804,C -0.3616,E1 18.2388,E2 604.7681} C_DIS
LIN {X -120.9932,Y -58.2847,Z 163,A -155.0039,B 18.3804,C -0.3591,E1 18.2402,E2 603.6321} C_DIS
LIN {X -119.0371,Y -62.1814,Z 163,A -153.159,B 18.3806,C -0.3535,E1 18.2425,E2 601.791} C_DIS
LIN {X -116.9098,Y -66.0987,Z 163,A -151.1579,B 18.3806,C -0.3521,E1 18.2452,E2 599.7798} C_DIS
LIN {X -114.6576,Y -69.9327,Z 163,A -149.2969,B 18.3806,C -0.3459,E1 18.2479,E2 597.9251} C_DIS
LIN {X -112.2235,Y -73.7748,Z 163,A -147.2994,B 18.3807,C -0.343,E1 18.2509,E2 595.9225} C_DIS
LIN {X -109.578,Y -77.6503,Z 163,A -145.3044,B 18.3808,C -0.3379,E1 18.2541,E2 593.9301} C_DIS
LIN {X -107.0113,Y -81.1511,Z 163,A -143.4665,B 18.3809,C -0.3329,E1 18.2571,E2 592.0956} C_DIS
LIN {X -104.3647,Y -84.5275,Z 163,A -141.573,B 18.3809,C -0.331,E1 18.2604,E2 590.1958} C_DIS
LIN {X -101.473,Y -87.9784,Z 163,A -139.9046,B 18.3812,C -0.3174,E1 18.2634,E2 588.56} C_DIS
LIN {X -98.9831,Y -90.77,Z 163,A -138.0355,B 18.3811,C -0.3239,E1 18.267,E2 586.6585} C_DIS
LIN {X -95.8974,Y -94.024,Z 163,A -136.1136,B 18.3811,C -0.3202,E1 18.2707,E2 584.7369} C_DIS
LIN {X -92.8228,Y -97.0605,Z 163,A -134.2946,B 18.3812,C -0.3155,E1 18.2743,E2 582.9221} C_DIS
LIN {X -89.7656,Y -99.895,Z 163,A -132.4759,B 18.3812,C -0.3135,E1 18.2781,E2 581.0996} C_DIS
LIN {X -86.6105,Y -102.6429,Z 163,A -130.8678,B 18.3814,C -0.3036,E1 18.2814,E2 579.5143} C_DIS
LIN {X -83.7695,Y -104.9739,Z 163,A -129.0876,B 18.3814,C -0.3086,E1 18.2854,E2 577.7088} C_DIS
LIN {X -80.1478,Y -107.7643,Z 163,A -127.1647,B 18.3814,C -0.3042,E1 18.2896,E2 575.7902} C_DIS
LIN {X -76.588,Y -110.3228,Z 163,A -125.2904,B 18.3814,C -0.3012,E1 18.2939,E2 573.9162} C_DIS
LIN {X -72.9405,Y -112.7677,Z 163,A -123.6554,B 18.3816,C -0.2894,E1 18.2976,E2 572.3114} C_DIS
LIN {X -68.1129,Y -115.7474,Z 163,A -120.9687,B 18.3816,C -0.2958,E1 18.3041,E2 569.5928} C_DIS
LIN {X -64.3575,Y -117.8768,Z 163,A -119.1044,B 18.3816,C -0.2941,E1 18.3087,E2 567.7262} C_DIS
LIN {X -60.9346,Y -119.6798,Z 163,A -117.5421,B 18.3816,C -0.2887,E1 18.3125,E2 566.1752} C_DIS
LIN {X -58.0072,Y -121.1258,Z 163,A -116.1525,B 18.3816,C -0.2869,E1 18.316,E2 564.7862} C_DIS
LIN {X -55.1163,Y -122.4687,Z 163,A -114.7461,B 18.3816,C -0.2871,E1 18.3196,E2 563.3743} C_DIS
LIN {X -51.8955,Y -123.8676,Z 163,A -113.2888,B 18.3817,C -0.284,E1 18.3233,E2 561.9222} C_DIS
LIN {X -48.6723,Y -125.1692,Z 163,A -111.8123,B 18.3817,C -0.2823,E1 18.3272,E2 560.4466} C_DIS
LIN {X -45.9785,Y -126.1844,Z 163,A -110.5439,B 18.3817,C -0.2827,E1 18.3305,E2 559.1734} C_DIS
LIN {X -42.6509,Y -127.3471,Z 163,A -108.9903,B 18.3817,C -0.2834,E1 18.3346,E2 557.6135} C_DIS
LIN {X -38.8888,Y -128.5464,Z 163,A -107.2295,B 18.3817,C -0.285,E1 18.3393,E2 555.8432} C_DIS
LIN {X -35.0754,Y -129.6391,Z 163,A -105.4676,B 18.3817,C -0.2866,E1 18.3441,E2 554.0725} C_DIS
LIN {X -30.5354,Y -130.7837,Z 163,A -103.5511,B 18.3817,C -0.2823,E1 18.3493,E2 552.1659} C_DIS
LIN {X -26.8749,Y -131.5831,Z 163,A -102.0496,B 18.3818,C -0.2779,E1 18.3533,E2 550.6761} C_DIS
LIN {X -23.8939,Y -132.1572,Z 163,A -100.6999,B 18.3818,C -0.2795,E1 18.3571,E2 549.3193} C_DIS
LIN {X -19.7701,Y -132.8388,Z 163,A -98.8529,B 18.3818,C -0.2814,E1 18.3622,E2 547.464} C_DIS
LIN {X -15.9337,Y -133.3511,Z 163,A -97.3169,B 18.3818,C -0.2766,E1 18.3664,E2 545.9417} C_DIS
LIN {X -12.0781,Y -133.7576,Z 163,A -95.5722,B 18.3818,C -0.2799,E1 18.3713,E2 544.1852} C_DIS
LIN {X -8.3164,Y -134.042,Z 163,A -93.998,B 18.3818,C -0.2785,E1 18.3757,E2 542.6147} C_DIS
LIN {X -3.9326,Y -134.2424,Z 163,A -92.1696,B 18.3818,C -0.2769,E1 18.3808,E2 540.7909} C_DIS
LIN {X -0.2069,Y -134.3008,Z 163,A -90.626,B 18.3818,C -0.2753,E1 18.3851,E2 539.2524} C_DIS
LIN {X -0.2069,Y -134.3008,Z 163,A -90.626,B 18.3818,C -0.2753,E1 18.3851,E2 539.2524} C_DIS
Enddeposition()
LIN {X 0.9356,Y -133.3729,Z 163,A -89.8941,B 17.1544,C -0.1472,E1 17.1572,E2 538.8576} C_DIS
Startdeposition()
$VEL.CP = VEL_PRINT
LIN {X -1.4856,Y -133.3727,Z 163,A -91.5913,B 17.1545,C -0.1233,E1 17.1523,E2 540.6358} C_DIS
LIN {X -5.48,Y -133.2666,Z 163,A -93.2152,B 17.1545,C -0.1265,E1 17.1478,E2 542.2491} C_DIS
LIN {X -9.574,Y -133.0348,Z 163,A -94.929,B 17.1545,C -0.1282,E1 17.143,E2 543.9579} C_DIS
LIN {X -13.2806,Y -132.7171,Z 163,A -96.4956,B 17.1545,C -0.1295,E1 17.1387,E2 545.5213} C_DIS
LIN {X -17.2798,Y -132.2547,Z 163,A -98.2527,B 17.1545,C -0.1289,E1 17.1338,E2 547.2822} C_DIS
LIN {X -21.1453,Y -131.694,Z 163,A -100.0547,B 17.1545,C -0.125,E1 17.1288,E2 549.0998} C_DIS
LIN {X -25.0084,Y -131.0131,Z 163,A -101.6162,B 17.1545,C -0.13,E1 17.1245,E2 550.6466} C_DIS
LIN {X -28.4918,Y -130.3004,Z 163,A -103.1583,B 17.1545,C -0.1302,E1 17.1203,E2 552.1908} C_DIS
LIN {X -35.2973,Y -128.6249,Z 163,A -106.0824,B 17.1545,C -0.135,E1 17.1124,E2 555.105} C_DIS
LIN {X -39.3791,Y -127.4333,Z 163,A -108.093,B 17.1545,C -0.1299,E1 17.107,E2 557.138} C_DIS
LIN {X -43.9735,Y -125.9216,Z 163,A -110.0616,B 17.1545,C -0.1354,E1 17.1018,E2 559.0933} C_DIS
LIN {X -47.3737,Y -124.6833,Z 163,A -111.6063,B 17.1545,C -0.1371,E1 17.0977,E2 560.6369} C_DIS
LIN {X -50.2081,Y -123.5681,Z 163,A -112.9327,B 17.1545,C -0.1378,E1 17.0943,E2 561.9654} C_DIS
LIN {X -53.2774,Y -122.2761,Z 163,A -114.3807,B 17.1545,C -0.1387,E1 17.0906,E2 563.4154} C_DIS
LIN {X -56.3939,Y -120.8707,Z 163,A -115.99,B 17.1545,C -0.1355,E1 17.0865,E2 565.0415} C_DIS
LIN {X -60.2575,Y -118.9911,Z 163,A -117.7161,B 17.1545,C -0.1419,E1 17.0822,E2 566.7528} C_DIS
LIN {X -63.6207,Y -117.2297,Z 163,A -119.4636,B 17.1545,C -0.14,E1 17.0778,E2 568.5141} C_DIS
LIN {X -67.4394,Y -115.075,Z 163,A -121.4908,B 17.1545,C -0.1377,E1 17.0729,E2 570.5581} C_DIS
Enddeposition()
END
